C05452=1014.580,211.144,368.499,168.044,54.073,160.186
C05453=1014.586,211.393,368.475,168.049,54.063,160.185
C05454=1014.591,211.642,368.450,168.054,54.053,160.184
C05455=1014.596,211.890,368.426,168.058,54.042,160.182
C05456=1014.601,212.139,368.401,168.063,54.032,160.181
C05457=1014.606,212.388,368.377,168.067,54.022,160.180
C05458=1014.613,212.637,368.352,168.072,54.012,160.179
C05459=1014.618,212.885,368.328,168.076,54.002,160.178
C05460=1014.622,213.134,368.303,168.081,53.992,160.176
C05461=1014.628,213.383,368.278,168.084,53.982,160.175
C05462=1014.633,213.631,368.254,168.089,53.972,160.174
C05463=1014.639,213.881,368.230,168.094,53.962,160.173
C05464=1014.644,214.129,368.205,168.098,53.952,160.172
C05465=1014.649,214.378,368.180,168.103,53.942,160.171
C05466=1014.654,214.626,368.155,168.108,53.932,160.169
C05467=1014.660,214.875,368.131,168.113,53.922,160.168
C05468=1014.666,215.124,368.107,168.116,53.913,160.167
C05469=1014.670,215.373,368.082,168.121,53.902,160.166
C05470=1014.676,215.622,368.057,168.126,53.892,160.165
C05471=1014.682,215.870,368.032,168.130,53.883,160.164
C05472=1014.687,216.119,368.008,168.135,53.872,160.162
C05473=1014.691,216.367,367.983,168.140,53.863,160.161
C05474=1014.697,216.617,367.958,168.144,53.853,160.160
C05475=1014.703,216.865,367.933,168.148,53.843,160.159
C05476=1014.708,217.113,367.909,168.153,53.833,160.158
C05477=1014.714,217.363,367.885,168.158,53.823,160.157
C05478=1014.719,217.612,367.860,168.163,53.814,160.156
C05479=1014.724,217.859,367.835,168.166,53.803,160.154
C05480=1014.730,218.108,367.810,168.171,53.794,160.153
C05481=1014.735,218.355,367.785,168.176,53.784,160.152
C05482=1014.740,218.600,367.761,168.179,53.775,160.151
C05483=1014.745,218.846,367.736,168.184,53.765,160.150
C05484=1014.750,219.092,367.711,168.188,53.756,160.149
C05485=1014.756,219.338,367.686,168.193,53.746,160.147
C05486=1014.761,219.584,367.660,168.197,53.737,160.147
C05487=1014.766,219.829,367.636,168.202,53.728,160.145
C05488=1014.771,220.075,367.611,168.206,53.718,160.144
C05489=1014.777,220.324,367.587,168.211,53.709,160.143
C05490=1014.782,220.573,367.561,168.216,53.699,160.142
C05491=1014.787,220.821,367.537,168.220,53.690,160.141
C05492=1014.793,221.070,367.511,168.225,53.680,160.140
C05493=1014.798,221.318,367.486,168.230,53.670,160.139
C05494=1014.803,221.568,367.461,168.234,53.661,160.138
C05495=1014.809,221.816,367.436,168.238,53.651,160.137
C05496=1014.814,222.065,367.410,168.243,53.641,160.136
C05497=1014.820,222.313,367.385,168.247,53.632,160.134
C05498=1014.825,222.562,367.360,168.252,53.622,160.133
C05499=1014.831,222.811,367.335,168.257,53.614,160.132
C05500=1014.835,223.059,367.310,168.261,53.604,160.131
C05501=1014.842,223.308,367.284,168.266,53.594,160.130
C05502=1014.846,223.557,367.260,168.270,53.585,160.129
C05503=1014.852,223.806,367.234,168.275,53.575,160.128
C05504=1014.857,224.054,367.209,168.279,53.566,160.127
C05505=1014.862,224.303,367.183,168.285,53.557,160.126
C05506=1014.868,224.551,367.158,168.288,53.548,160.125
C05507=1014.873,224.800,367.132,168.293,53.538,160.124
C05508=1014.880,225.049,367.107,168.298,53.528,160.123
C05509=1014.884,225.298,367.082,168.303,53.520,160.122
C05510=1014.890,225.547,367.057,168.308,53.510,160.121
C05511=1014.895,225.795,367.031,168.312,53.501,160.120
C05512=1014.902,226.044,367.006,168.317,53.492,160.119
C05513=1014.906,226.292,366.980,168.321,53.483,160.118
C05514=1014.912,226.541,366.955,168.326,53.473,160.117
C05515=1014.916,226.790,366.930,168.330,53.464,160.116
C05516=1014.922,227.039,366.904,168.335,53.455,160.115
C05517=1014.928,227.287,366.878,168.340,53.446,160.114
C05518=1014.933,227.536,366.853,168.343,53.437,160.112
C05519=1014.938,227.785,366.827,168.349,53.428,160.112
C05520=1014.943,228.033,366.801,168.353,53.419,160.110
C05521=1014.949,228.282,366.776,168.358,53.410,160.110
C05522=1014.955,228.531,366.750,168.362,53.400,160.108
C05523=1014.960,228.779,366.725,168.368,53.392,160.108
C05524=1014.965,229.028,366.699,168.372,53.382,160.106
C05525=1014.970,229.276,366.673,168.376,53.374,160.105
C05526=1014.977,229.524,366.647,168.381,53.365,160.105
C05527=1014.982,229.773,366.621,168.385,53.355,160.103
C05528=1014.987,230.021,366.595,168.391,53.347,160.103
C05529=1014.992,230.270,366.570,168.395,53.338,160.102
C05530=1014.998,230.519,366.544,168.399,53.329,160.101
C05531=1015.003,230.768,366.518,168.405,53.320,160.100
C05532=1015.009,231.016,366.491,168.409,53.311,160.099
C05533=1015.014,231.265,366.465,168.413,53.303,160.098
C05534=1015.019,231.513,366.440,168.418,53.293,160.097
C05535=1015.024,231.762,366.414,168.423,53.284,160.096
C05536=1015.030,232.011,366.388,168.427,53.276,160.095
C05537=1015.035,232.259,366.362,168.432,53.267,160.094
C05538=1015.040,232.508,366.336,168.437,53.258,160.093
C05539=1015.046,232.757,366.310,168.441,53.249,160.092
C05540=1015.051,233.004,366.284,168.445,53.241,160.091
C05541=1015.057,233.246,366.258,168.450,53.232,160.090
C05542=1015.062,233.488,366.233,168.454,53.224,160.089
C05543=1015.068,233.730,366.208,168.460,53.215,160.088
C05544=1015.072,233.972,366.182,168.465,53.207,160.088
C05545=1015.078,234.213,366.157,168.469,53.198,160.087
C05546=1015.083,234.455,366.132,168.474,53.190,160.086
C05547=1015.089,234.697,366.107,168.478,53.181,160.085
C05548=1015.094,234.938,366.082,168.483,53.173,160.084
C05549=1015.100,235.187,366.055,168.487,53.164,160.083
C05550=1015.105,235.436,366.029,168.491,53.156,160.082
C05551=1015.111,235.684,366.003,168.497,53.147,160.081
C05552=1015.116,235.933,365.977,168.501,53.138,160.080
C05553=1015.121,236.181,365.951,168.506,53.130,160.079
C05554=1015.127,236.430,365.925,168.510,53.121,160.078
C05555=1015.132,236.679,365.899,168.515,53.113,160.077
C05556=1015.138,236.927,365.872,168.520,53.104,160.076
C05557=1015.144,237.176,365.846,168.525,53.095,160.076
C05558=1015.149,237.424,365.819,168.530,53.087,160.075
C05559=1015.154,237.673,365.794,168.534,53.079,160.074
C05560=1015.159,237.921,365.767,168.538,53.070,160.073
C05561=1015.165,238.170,365.740,168.544,53.061,160.072
C05562=1015.171,238.419,365.714,168.548,53.053,160.071
C05563=1015.176,238.667,365.687,168.553,53.044,160.070
C05564=1015.182,238.915,365.661,168.558,53.037,160.070
C05565=1015.187,239.164,365.635,168.562,53.028,160.069
C05566=1015.193,239.412,365.608,168.567,53.020,160.068
C05567=1015.198,239.661,365.581,168.572,53.012,160.067
C05568=1015.204,239.909,365.555,168.576,53.003,160.066
C05569=1015.209,240.158,365.529,168.582,52.994,160.065
C05570=1015.214,240.407,365.501,168.587,52.987,160.064
C05571=1015.220,240.655,365.475,168.591,52.978,160.064
C05572=1015.226,240.903,365.448,168.596,52.970,160.063
C05573=1015.230,241.153,365.422,168.600,52.962,160.062
C05574=1015.236,241.401,365.395,168.605,52.953,160.061
C05575=1015.242,241.649,365.368,168.610,52.946,160.060
C05576=1015.248,241.898,365.342,168.614,52.937,160.059
C05577=1015.253,242.146,365.314,168.619,52.929,160.059
C05578=1015.258,242.394,365.288,168.624,52.921,160.058
C05579=1015.264,242.642,365.261,168.629,52.913,160.057
C05580=1015.269,242.891,365.234,168.633,52.905,160.056
C05581=1015.275,243.139,365.208,168.638,52.897,160.055
C05582=1015.280,243.388,365.180,168.643,52.888,160.054
C05583=1015.285,243.636,365.154,168.648,52.880,160.054
C05584=1015.290,243.885,365.126,168.653,52.873,160.053
C05585=1015.295,244.134,365.099,168.657,52.864,160.052
C05586=1015.301,244.382,365.073,168.662,52.856,160.051
C05587=1015.306,244.631,365.045,168.667,52.849,160.051
C05588=1015.312,244.879,365.019,168.672,52.841,160.050
C05589=1015.317,245.127,364.991,168.676,52.832,160.049
C05590=1015.322,245.376,364.963,168.681,52.825,160.048
C05591=1015.328,245.624,364.937,168.686,52.817,160.047
C05592=1015.333,245.873,364.910,168.691,52.809,160.047
C05593=1015.339,246.121,364.883,168.696,52.801,160.046
C05594=1015.344,246.370,364.856,168.701,52.793,160.045
C05595=1015.350,246.619,364.827,168.705,52.785,160.044
C05596=1015.356,246.867,364.801,168.710,52.778,160.044
C05597=1015.361,247.116,364.773,168.715,52.770,160.043
C05598=1015.367,247.364,364.747,168.719,52.761,160.042
C05599=1015.372,247.612,364.719,168.724,52.754,160.041
C05600=1015.378,247.861,364.692,168.729,52.746,160.040
C05601=1015.383,248.098,364.666,168.734,52.738,160.040
C05602=1015.388,248.338,364.640,168.739,52.731,160.039
C05603=1015.393,248.576,364.614,168.743,52.724,160.038
C05604=1015.398,248.814,364.588,168.747,52.716,160.038
C05605=1015.404,249.052,364.561,168.752,52.708,160.037
C05606=1015.409,249.290,364.535,168.756,52.701,160.036
C05607=1015.414,249.529,364.508,168.762,52.694,160.036
C05608=1015.419,249.768,364.483,168.767,52.686,160.035
C05609=1015.425,250.015,364.455,168.771,52.679,160.034
C05610=1015.430,250.264,364.428,168.776,52.671,160.033
C05611=1015.437,250.512,364.400,168.781,52.663,160.033
C05612=1015.442,250.761,364.373,168.786,52.656,160.032
C05613=1015.447,251.010,364.346,168.791,52.648,160.031
C05614=1015.453,251.257,364.319,168.796,52.640,160.030
C05615=1015.458,251.506,364.291,168.801,52.632,160.030
C05616=1015.465,251.755,364.264,168.806,52.625,160.029
C05617=1015.470,252.003,364.236,168.810,52.617,160.028
C05618=1015.475,252.251,364.208,168.815,52.610,160.027
C05619=1015.481,252.500,364.182,168.820,52.602,160.027
C05620=1015.487,252.748,364.153,168.825,52.595,160.026
C05621=1015.493,252.997,364.127,168.830,52.587,160.026
C05622=1015.498,253.245,364.099,168.835,52.579,160.025
C05623=1015.504,253.494,364.071,168.840,52.572,160.024
C05624=1015.510,253.742,364.044,168.844,52.564,160.023
C05625=1015.515,253.991,364.017,168.849,52.556,160.023
C05626=1015.521,254.239,363.988,168.854,52.549,160.022
C05627=1015.527,254.488,363.962,168.859,52.542,160.021
C05628=1015.532,254.736,363.934,168.864,52.534,160.021
C05629=1015.539,254.984,363.906,168.869,52.526,160.020
C05630=1015.544,255.233,363.879,168.874,52.519,160.019
C05631=1015.549,255.481,363.851,168.879,52.512,160.019
C05632=1015.555,255.730,363.824,168.884,52.504,160.018
C05633=1015.561,255.978,363.796,168.889,52.496,160.017
C05634=1015.567,256.226,363.768,168.894,52.489,160.017
C05635=1015.572,256.475,363.741,168.899,52.482,160.016
C05636=1015.578,256.723,363.713,168.903,52.474,160.015
C05637=1015.584,256.972,363.685,168.909,52.467,160.015
C05638=1015.590,257.220,363.657,168.914,52.460,160.014
C05639=1015.595,257.469,363.630,168.919,52.452,160.013
C05640=1015.601,257.717,363.602,168.924,52.445,160.013
C05641=1015.607,257.965,363.574,168.929,52.437,160.012
C05642=1015.613,258.213,363.546,168.933,52.430,160.011
C05643=1015.618,258.462,363.519,168.939,52.423,160.011
C05644=1015.624,258.711,363.491,168.944,52.415,160.010
C05645=1015.631,258.958,363.464,168.949,52.408,160.009
C05646=1015.636,259.207,363.435,168.954,52.400,160.009
C05647=1015.643,259.455,363.408,168.959,52.394,160.008
C05648=1015.648,259.703,363.380,168.964,52.386,160.007
C05649=1015.654,259.952,363.352,168.969,52.379,160.007
C05650=1015.659,260.200,363.324,168.974,52.372,160.006
C05651=1015.665,260.449,363.295,168.979,52.365,160.006
C05652=1015.670,260.697,363.267,168.984,52.358,160.005
C05653=1015.676,260.945,363.239,168.988,52.351,160.004
C05654=1015.682,261.193,363.211,168.994,52.343,160.004
C05655=1015.688,261.442,363.182,168.999,52.336,160.003
C05656=1015.693,261.690,363.154,169.003,52.330,160.003
C05657=1015.699,261.938,363.126,169.009,52.323,160.002
C05658=1015.704,262.187,363.097,169.014,52.315,160.001
C05659=1015.710,262.435,363.069,169.018,52.308,160.001
C05660=1015.715,262.683,363.041,169.024,52.301,160.000
C05661=1015.721,262.921,363.014,169.028,52.295,160.000
C05662=1015.727,263.158,362.986,169.034,52.288,159.999
C05663=1015.732,263.396,362.959,169.038,52.281,159.999
C05664=1015.737,263.633,362.932,169.043,52.274,159.998
C05665=1015.743,263.870,362.905,169.049,52.268,159.998
C05666=1015.748,264.108,362.878,169.053,52.261,159.997
C05667=1015.754,264.345,362.851,169.058,52.255,159.997
C05668=1015.760,264.582,362.823,169.063,52.248,159.996
C05669=1015.765,264.830,362.795,169.067,52.241,159.995
C05670=1015.771,265.079,362.767,169.073,52.234,159.995
C05671=1015.777,265.326,362.738,169.077,52.228,159.994
C05672=1015.783,265.575,362.710,169.083,52.221,159.994
C05673=1015.788,265.824,362.680,169.088,52.214,159.993
C05674=1015.794,266.072,362.652,169.093,52.207,159.993
C05675=1015.799,266.320,362.624,169.098,52.200,159.992
C05676=1015.806,266.569,362.595,169.103,52.193,159.992
C05677=1015.811,266.817,362.567,169.108,52.186,159.991
C05678=1015.817,267.065,362.537,169.114,52.179,159.991
C05679=1015.823,267.314,362.509,169.119,52.173,159.990
C05680=1015.828,267.561,362.480,169.124,52.166,159.990
C05681=1015.834,267.810,362.452,169.129,52.160,159.989
C05682=1015.840,268.058,362.423,169.134,52.153,159.989
C05683=1015.846,268.307,362.393,169.140,52.146,159.988
C05684=1015.851,268.555,362.365,169.144,52.139,159.987
C05685=1015.857,268.803,362.336,169.150,52.132,159.987
C05686=1015.863,269.052,362.308,169.154,52.126,159.987
C05687=1015.868,269.299,362.279,169.160,52.119,159.986
C05688=1015.875,269.547,362.250,169.164,52.113,159.985
C05689=1015.880,269.796,362.220,169.170,52.106,159.985
C05690=1015.886,270.045,362.192,169.175,52.100,159.985
C05691=1015.892,270.292,362.163,169.180,52.093,159.984
C05692=1015.897,270.540,362.133,169.185,52.087,159.984
C05693=1015.903,270.789,362.104,169.191,52.080,159.983
C05694=1015.909,271.037,362.076,169.196,52.073,159.983
C05695=1015.915,271.286,362.046,169.201,52.067,159.982
C05696=1015.921,271.533,362.018,169.207,52.060,159.982
C05697=1015.926,271.782,361.988,169.211,52.054,159.981
C05698=1015.932,272.030,361.959,169.217,52.047,159.981
C05699=1015.939,272.278,361.930,169.222,52.041,159.980
C05700=1015.944,272.527,361.901,169.228,52.034,159.980
C05701=1015.949,272.774,361.872,169.232,52.028,159.979
C05702=1015.955,273.023,361.843,169.238,52.021,159.979
C05703=1015.961,273.271,361.814,169.242,52.015,159.978
C05704=1015.967,273.519,361.784,169.248,52.009,159.978
C05705=1015.973,273.768,361.755,169.253,52.002,159.978
C05706=1015.978,274.016,361.725,169.259,51.996,159.977
C05707=1015.985,274.264,361.696,169.264,51.990,159.977
C05708=1015.990,274.513,361.667,169.269,51.983,159.976
C05709=1015.996,274.761,361.638,169.274,51.977,159.976
C05710=1016.001,275.008,361.609,169.280,51.970,159.975
C05711=1016.008,275.257,361.579,169.285,51.964,159.975
C05712=1016.013,275.505,361.550,169.291,51.958,159.975
C05713=1016.020,275.753,361.520,169.295,51.951,159.974
C05714=1016.026,276.001,361.491,169.301,51.945,159.974
C05715=1016.031,276.249,361.461,169.306,51.939,159.974
C05716=1016.037,276.498,361.432,169.310,51.933,159.973
C05717=1016.043,276.746,361.403,169.316,51.926,159.973
C05718=1016.049,276.994,361.372,169.321,51.920,159.972
C05719=1016.054,277.242,361.343,169.327,51.914,159.972
C05720=1016.060,277.490,361.313,169.332,51.908,159.972
C05721=1016.066,277.729,361.285,169.337,51.902,159.971
C05722=1016.071,277.970,361.256,169.342,51.896,159.971
C05723=1016.077,278.209,361.227,169.348,51.890,159.970
C05724=1016.082,278.448,361.198,169.353,51.884,159.970
C05725=1016.089,278.688,361.170,169.358,51.878,159.970
C05726=1016.094,278.927,361.141,169.363,51.872,159.969
C05727=1016.100,279.167,361.112,169.368,51.867,159.969
C05728=1016.105,279.406,361.084,169.373,51.861,159.968
C05729=1016.111,279.655,361.054,169.379,51.854,159.968
C05730=1016.117,279.903,361.024,169.383,51.849,159.968
C05731=1016.123,280.151,360.994,169.389,51.842,159.967
C05732=1016.129,280.399,360.964,169.394,51.836,159.967
C05733=1016.134,280.647,360.934,169.400,51.830,159.967
C05734=1016.141,280.895,360.904,169.405,51.824,159.966
C05735=1016.147,281.144,360.875,169.410,51.818,159.966
C05736=1016.153,281.391,360.844,169.416,51.812,159.966
C05737=1016.158,281.640,360.815,169.421,51.806,159.965
C05738=1016.165,281.887,360.785,169.427,51.800,159.965
C05739=1016.170,282.136,360.755,169.432,51.794,159.965
C05740=1016.176,282.384,360.725,169.437,51.788,159.964
C05741=1016.182,282.633,360.695,169.443,51.783,159.964
C05742=1016.189,282.880,360.665,169.448,51.777,159.964
C05743=1016.195,283.128,360.635,169.454,51.771,159.963
C05744=1016.200,283.377,360.605,169.459,51.765,159.963
C05745=1016.206,283.624,360.575,169.465,51.758,159.963
C05746=1016.212,283.872,360.545,169.470,51.753,159.962
C05747=1016.219,284.121,360.515,169.475,51.747,159.962
C05748=1016.224,284.369,360.485,169.481,51.741,159.962
C05749=1016.230,284.617,360.454,169.486,51.735,159.961
C05750=1016.236,284.865,360.424,169.492,51.729,159.961
C05751=1016.242,285.114,360.394,169.498,51.724,159.961
C05752=1016.248,285.361,360.364,169.503,51.718,159.961
C05753=1016.254,285.609,360.333,169.508,51.712,159.960
C05754=1016.260,285.857,360.304,169.514,51.707,159.960
C05755=1016.267,286.105,360.273,169.519,51.701,159.960
C05756=1016.273,286.353,360.243,169.525,51.695,159.960
C05757=1016.278,286.601,360.212,169.530,51.689,159.959
C05758=1016.284,286.849,360.182,169.535,51.683,159.959
C05759=1016.291,287.097,360.151,169.541,51.678,159.959
C05760=1016.296,287.345,360.121,169.546,51.672,159.958
C05761=1016.302,287.593,360.090,169.552,51.667,159.958
C05762=1016.309,287.841,360.060,169.558,51.661,159.958
C05763=1016.315,288.089,360.029,169.563,51.655,159.958
C05764=1016.320,288.337,359.999,169.568,51.650,159.957
C05765=1016.326,288.586,359.968,169.574,51.644,159.957
C05766=1016.332,288.834,359.937,169.579,51.638,159.957
C05767=1016.338,289.082,359.907,169.586,51.633,159.957
C05768=1016.344,289.330,359.876,169.591,51.627,159.957
C05769=1016.350,289.578,359.846,169.596,51.622,159.956
C05770=1016.356,289.825,359.815,169.602,51.616,159.956
C05771=1016.362,290.074,359.784,169.607,51.610,159.956
C05772=1016.368,290.321,359.754,169.613,51.605,159.955
C05773=1016.375,290.570,359.723,169.619,51.599,159.955
C05774=1016.380,290.818,359.693,169.624,51.594,159.955
C05775=1016.387,291.065,359.662,169.630,51.588,159.955
C05776=1016.393,291.314,359.631,169.636,51.583,159.955
C05777=1016.398,291.562,359.600,169.641,51.578,159.955
C05778=1016.405,291.810,359.569,169.646,51.572,159.954
C05779=1016.411,292.057,359.538,169.653,51.566,159.954
C05780=1016.417,292.306,359.508,169.658,51.561,159.954
C05781=1016.423,292.551,359.477,169.663,51.556,159.954
C05782=1016.429,292.797,359.446,169.669,51.551,159.953
C05783=1016.435,293.043,359.416,169.675,51.545,159.953
C05784=1016.441,293.289,359.384,169.681,51.540,159.953
C05785=1016.446,293.534,359.353,169.686,51.535,159.953
C05786=1016.453,293.779,359.322,169.691,51.530,159.953
C05787=1016.458,294.026,359.292,169.697,51.524,159.953
C05788=1016.464,294.272,359.260,169.702,51.519,159.952
C05789=1016.470,294.519,359.229,169.708,51.514,159.952
C05790=1016.476,294.767,359.197,169.714,51.509,159.952
C05791=1016.482,295.015,359.167,169.719,51.503,159.952
C05792=1016.488,295.263,359.135,169.725,51.498,159.952
C05793=1016.493,295.511,359.103,169.731,51.493,159.952
C05794=1016.500,295.759,359.072,169.736,51.488,159.951
C05795=1016.505,296.007,359.041,169.742,51.482,159.951
C05796=1016.512,296.255,359.009,169.748,51.478,159.951
C05797=1016.518,296.503,358.977,169.754,51.472,159.951
C05798=1016.524,296.750,358.946,169.759,51.467,159.951
C05799=1016.530,296.999,358.915,169.765,51.462,159.951
C05800=1016.536,297.246,358.884,169.770,51.457,159.951
C05801=1016.542,297.494,358.852,169.777,51.452,159.951
C05802=1016.549,297.742,358.820,169.782,51.447,159.951
C05803=1016.554,297.990,358.789,169.788,51.442,159.950
C05804=1016.561,298.238,358.757,169.793,51.437,159.950
C05805=1016.567,298.486,358.725,169.799,51.431,159.950
C05806=1016.572,298.733,358.694,169.805,51.427,159.950
C05807=1016.579,298.981,358.662,169.811,51.421,159.950
C05808=1016.585,299.229,358.630,169.816,51.416,159.950
C05809=1016.591,299.477,358.599,169.823,51.411,159.950
C05810=1016.597,299.725,358.567,169.828,51.406,159.950
C05811=1016.604,299.973,358.536,169.834,51.401,159.949
C05812=1016.610,300.221,358.504,169.840,51.396,159.950
C05813=1016.616,300.468,358.472,169.846,51.391,159.949
C05814=1016.622,300.716,358.440,169.852,51.387,159.949
C05815=1016.628,300.964,358.409,169.857,51.381,159.949
C05816=1016.634,301.212,358.377,169.863,51.376,159.949
C05817=1016.640,301.460,358.345,169.869,51.371,159.949
C05818=1016.647,301.708,358.314,169.875,51.366,159.949
C05819=1016.653,301.956,358.282,169.880,51.362,159.949
C05820=1016.659,302.204,358.250,169.887,51.356,159.949
C05821=1016.665,302.452,358.218,169.893,51.352,159.949
C05822=1016.672,302.699,358.187,169.898,51.347,159.949
C05823=1016.678,302.947,358.155,169.905,51.342,159.949
C05824=1016.684,303.195,358.123,169.910,51.337,159.949
C05825=1016.690,303.443,358.091,169.916,51.332,159.949
C05826=1016.697,303.690,358.059,169.921,51.327,159.948
C05827=1016.703,303.939,358.027,169.928,51.322,159.949
C05828=1016.709,304.187,357.995,169.934,51.318,159.949
C05829=1016.716,304.435,357.963,169.939,51.313,159.948
C05830=1016.722,304.682,357.931,169.946,51.308,159.948
C05831=1016.729,304.929,357.900,169.952,51.303,159.948
C05832=1016.735,305.178,357.868,169.957,51.298,159.948
C05833=1016.742,305.425,357.835,169.963,51.294,159.948
C05834=1016.748,305.673,357.803,169.970,51.288,159.948
C05835=1016.755,305.920,357.771,169.975,51.284,159.948
C05836=1016.761,306.169,357.739,169.981,51.279,159.948
C05837=1016.767,306.417,357.707,169.988,51.274,159.948
C05838=1016.774,306.664,357.675,169.993,51.269,159.948
C05839=1016.780,306.912,357.643,169.999,51.265,159.948
C05840=1016.787,307.160,357.611,170.005,51.260,159.948
C05841=1016.793,307.422,357.577,170.011,51.255,159.948
C05842=1016.800,307.682,357.543,170.018,51.250,159.948
C05843=1016.807,307.944,357.509,170.025,51.245,159.948
C05844=1016.814,308.206,357.475,170.030,51.240,159.948
C05845=1016.821,308.453,357.443,170.037,51.235,159.948
C05846=1016.827,308.701,357.410,170.043,51.231,159.948
C05847=1016.834,308.949,357.379,170.049,51.226,159.948
C05848=1016.840,309.196,357.346,170.056,51.221,159.948
C05849=1016.847,309.444,357.315,170.061,51.217,159.948
C05850=1016.853,309.692,357.282,170.067,51.212,159.948
C05851=1016.859,309.940,357.248,170.073,51.208,159.948
C05852=1016.865,310.187,357.216,170.080,51.203,159.948
C05853=1016.871,310.435,357.183,170.086,51.199,159.948
C05854=1016.878,310.683,357.150,170.092,51.194,159.948
C05855=1016.884,310.930,357.118,170.098,51.190,159.949
C05856=1016.890,311.179,357.084,170.104,51.186,159.949
C05857=1016.896,311.426,357.051,170.109,51.182,159.949
C05858=1016.903,311.674,357.018,170.116,51.177,159.949
C05859=1016.909,311.921,356.985,170.122,51.173,159.949
C05860=1016.916,312.169,356.952,170.128,51.168,159.949
C05861=1016.921,312.416,356.919,170.134,51.164,159.949
C05862=1016.928,312.664,356.886,170.140,51.159,159.949
C05863=1016.934,312.912,356.853,170.147,51.155,159.949
C05864=1016.941,313.160,356.820,170.153,51.151,159.949
C05865=1016.947,313.408,356.787,170.159,51.147,159.950
C05866=1016.953,313.655,356.753,170.165,51.143,159.950
C05867=1016.959,313.902,356.721,170.172,51.138,159.950
C05868=1016.966,314.151,356.688,170.178,51.134,159.950
C05869=1016.972,314.398,356.655,170.184,51.130,159.950
C05870=1016.979,314.645,356.621,170.190,51.126,159.950
C05871=1016.984,314.893,356.588,170.196,51.121,159.950
C05872=1016.991,315.141,356.555,170.203,51.116,159.950
C05873=1016.998,315.388,356.521,170.209,51.113,159.950
C05874=1017.004,315.636,356.489,170.215,51.108,159.950
C05875=1017.011,315.884,356.456,170.221,51.104,159.951
C05876=1017.017,316.132,356.422,170.228,51.100,159.951
C05877=1017.023,316.379,356.389,170.234,51.096,159.951
C05878=1017.031,316.627,356.355,170.240,51.092,159.951
C05879=1017.037,316.874,356.322,170.246,51.088,159.951
C05880=1017.043,317.123,356.289,170.253,51.083,159.952
C05881=1017.050,317.370,356.255,170.259,51.079,159.952
C05882=1017.056,317.618,356.222,170.265,51.075,159.952
C05883=1017.063,317.865,356.188,170.271,51.071,159.952
C05884=1017.069,318.113,356.156,170.278,51.067,159.952
C05885=1017.076,318.361,356.121,170.284,51.063,159.952
C05886=1017.082,318.609,356.089,170.290,51.058,159.952
C05887=1017.089,318.856,356.055,170.297,51.054,159.953
C05888=1017.096,319.103,356.021,170.304,51.050,159.953
C05889=1017.102,319.352,355.988,170.310,51.047,159.953
C05890=1017.109,319.599,355.954,170.316,51.042,159.953
C05891=1017.116,319.846,355.920,170.323,51.038,159.953
C05892=1017.122,320.094,355.888,170.329,51.034,159.954
C05893=1017.129,320.342,355.854,170.335,51.030,159.954
C05894=1017.135,320.589,355.820,170.341,51.026,159.954
C05895=1017.142,320.837,355.787,170.348,51.022,159.954
C05896=1017.149,321.085,355.753,170.355,51.018,159.954
C05897=1017.156,321.332,355.719,170.361,51.014,159.954
C05898=1017.162,321.580,355.685,170.368,51.010,159.955
C05899=1017.169,321.827,355.652,170.374,51.006,159.955
C05900=1017.176,322.075,355.618,170.380,51.002,159.955
C05901=1017.183,322.342,355.581,170.387,50.998,159.955
C05902=1017.190,322.608,355.545,170.394,50.994,159.956
C05903=1017.198,322.875,355.509,170.402,50.989,159.956
C05904=1017.205,323.142,355.473,170.409,50.985,159.956
C05905=1017.212,323.389,355.439,170.415,50.981,159.956
C05906=1017.219,323.638,355.406,170.421,50.978,159.957
C05907=1017.225,323.885,355.372,170.429,50.974,159.957
C05908=1017.232,324.133,355.338,170.435,50.970,159.957
C05909=1017.239,324.380,355.304,170.441,50.966,159.957
C05910=1017.246,324.628,355.270,170.448,50.962,159.958
C05911=1017.253,324.876,355.236,170.454,50.958,159.958
C05912=1017.260,325.123,355.202,170.461,50.954,159.958
C05913=1017.267,325.371,355.168,170.468,50.950,159.958
C05914=1017.274,325.618,355.135,170.474,50.946,159.959
C05915=1017.281,325.866,355.099,170.480,50.943,159.959
C05916=1017.288,326.113,355.066,170.488,50.939,159.959
C05917=1017.295,326.360,355.032,170.494,50.935,159.960
C05918=1017.301,326.608,354.998,170.500,50.931,159.960
C05919=1017.308,326.856,354.963,170.508,50.927,159.960
C05920=1017.315,327.103,354.929,170.514,50.924,159.960
C05921=1017.321,327.351,354.894,170.520,50.920,159.961
C05922=1017.328,327.599,354.859,170.528,50.917,159.961
C05923=1017.335,327.846,354.826,170.534,50.913,159.961
C05924=1017.342,328.093,354.791,170.540,50.909,159.962
C05925=1017.348,328.341,354.756,170.547,50.906,159.962
C05926=1017.356,328.588,354.722,170.554,50.902,159.962
C05927=1017.362,328.836,354.687,170.561,50.899,159.963
C05928=1017.369,329.083,354.652,170.567,50.895,159.963
C05929=1017.375,329.331,354.618,170.575,50.892,159.963
C05930=1017.383,329.578,354.583,170.581,50.888,159.964
C05931=1017.389,329.826,354.549,170.588,50.885,159.964
C05932=1017.396,330.074,354.514,170.595,50.881,159.964
C05933=1017.403,330.321,354.479,170.601,50.878,159.965
C05934=1017.410,330.569,354.445,170.608,50.874,159.965
C05935=1017.417,330.816,354.409,170.615,50.870,159.965
C05936=1017.424,331.063,354.375,170.622,50.867,159.966
C05937=1017.431,331.311,354.341,170.629,50.864,159.966
C05938=1017.437,331.559,354.305,170.636,50.860,159.967
C05939=1017.444,331.806,354.270,170.642,50.857,159.967
C05940=1017.451,332.054,354.236,170.649,50.854,159.967
C05941=1017.458,332.301,354.201,170.656,50.850,159.968
C05942=1017.465,332.548,354.166,170.663,50.846,159.968
C05943=1017.472,332.796,354.131,170.669,50.843,159.969
C05944=1017.478,333.043,354.096,170.677,50.840,159.969
C05945=1017.487,333.291,354.061,170.684,50.837,159.969
C05946=1017.493,333.538,354.026,170.690,50.833,159.970
C05947=1017.500,333.786,353.991,170.698,50.829,159.970
C05948=1017.507,334.033,353.956,170.704,50.826,159.971
C05949=1017.514,334.280,353.920,170.711,50.823,159.971
C05950=1017.520,334.528,353.885,170.718,50.820,159.971
C05951=1017.527,334.775,353.850,170.725,50.817,159.972
C05952=1017.535,335.023,353.815,170.732,50.813,159.972
C05953=1017.541,335.270,353.780,170.739,50.810,159.973
C05954=1017.548,335.517,353.744,170.746,50.807,159.973
C05955=1017.555,335.765,353.709,170.752,50.804,159.974
C05956=1017.563,336.013,353.673,170.760,50.800,159.974
C05957=1017.569,336.260,353.638,170.767,50.797,159.975
C05958=1017.576,336.507,353.603,170.773,50.794,159.975
C05959=1017.583,336.754,353.567,170.781,50.790,159.975
C05960=1017.590,337.002,353.531,170.788,50.787,159.976
C05961=1017.598,337.265,353.494,170.796,50.785,159.977
C05962=1017.606,337.527,353.457,170.803,50.781,159.977
C05963=1017.613,337.790,353.419,170.811,50.778,159.978
C05964=1017.620,338.052,353.381,170.818,50.774,159.978
C05965=1017.627,338.300,353.346,170.825,50.771,159.978
C05966=1017.635,338.547,353.310,170.832,50.768,159.979
C05967=1017.642,338.795,353.274,170.840,50.765,159.980
C05968=1017.649,339.042,353.238,170.846,50.762,159.980
C05969=1017.656,339.289,353.203,170.854,50.758,159.981
C05970=1017.663,339.536,353.167,170.861,50.756,159.981
C05971=1017.671,339.783,353.131,170.868,50.753,159.982
C05972=1017.678,340.031,353.096,170.875,50.749,159.982
C05973=1017.684,340.278,353.059,170.882,50.747,159.983
C05974=1017.691,340.526,353.024,170.890,50.743,159.983
C05975=1017.699,340.773,352.988,170.897,50.741,159.984
C05976=1017.706,341.020,352.952,170.903,50.738,159.984
C05977=1017.713,341.267,352.916,170.911,50.735,159.985
C05978=1017.719,341.515,352.880,170.918,50.732,159.985
C05979=1017.727,341.762,352.844,170.926,50.729,159.986
C05980=1017.734,342.009,352.808,170.933,50.726,159.986
C05981=1017.742,342.256,352.772,170.941,50.723,159.987
C05982=1017.748,342.504,352.735,170.947,50.720,159.988
C05983=1017.756,342.751,352.699,170.954,50.717,159.988
C05984=1017.764,342.998,352.663,170.962,50.715,159.989
C05985=1017.771,343.245,352.627,170.969,50.711,159.989
C05986=1017.778,343.493,352.590,170.977,50.709,159.990
C05987=1017.785,343.740,352.554,170.984,50.706,159.991
C05988=1017.792,343.987,352.518,170.992,50.703,159.991
C05989=1017.799,344.235,352.481,170.999,50.700,159.992
C05990=1017.806,344.482,352.445,171.007,50.697,159.992
C05991=1017.814,344.729,352.409,171.014,50.695,159.993
C05992=1017.821,344.977,352.372,171.021,50.692,159.994
C05993=1017.828,345.224,352.337,171.028,50.689,159.994
C05994=1017.836,345.471,352.300,171.035,50.686,159.995
C05995=1017.843,345.719,352.264,171.043,50.684,159.995
C05996=1017.850,345.966,352.227,171.050,50.681,159.996
C05997=1017.858,346.212,352.191,171.058,50.678,159.997
C05998=1017.865,346.460,352.155,171.065,50.676,159.997
C05999=1017.872,346.708,352.118,171.073,50.673,159.998
C06000=1017.880,346.954,352.081,171.080,50.671,159.999
C06001=1017.887,347.201,352.044,171.088,50.668,159.999
C06002=1017.894,347.449,352.008,171.095,50.665,160.000
C06003=1017.902,347.696,351.971,171.103,50.662,160.001
C06004=1017.909,347.943,351.934,171.110,50.660,160.001
C06005=1017.916,348.191,351.897,171.118,50.657,160.002
C06006=1017.924,348.438,351.861,171.125,50.655,160.003
C06007=1017.931,348.684,351.824,171.133,50.652,160.003
C06008=1017.938,348.932,351.787,171.140,50.649,160.004
C06009=1017.946,349.179,351.750,171.149,50.647,160.005
C06010=1017.953,349.426,351.712,171.156,50.645,160.005
C06011=1017.961,349.674,351.676,171.164,50.642,160.006
C06012=1017.968,349.921,351.639,171.172,50.639,160.007
C06013=1017.976,350.168,351.602,171.179,50.637,160.008
C06014=1017.983,350.415,351.565,171.187,50.634,160.008
C06015=1017.991,350.662,351.528,171.194,50.632,160.009
C06016=1017.998,350.909,351.490,171.202,50.629,160.010
C06017=1018.005,351.156,351.453,171.210,50.627,160.011
C06018=1018.013,351.404,351.417,171.218,50.624,160.011
C06019=1018.020,351.651,351.379,171.225,50.622,160.012
C06020=1018.028,351.898,351.342,171.233,50.620,160.013
C06021=1018.036,352.158,351.303,171.241,50.617,160.013
C06022=1018.044,352.417,351.264,171.249,50.615,160.014
C06023=1018.052,352.677,351.225,171.257,50.612,160.015
C06024=1018.060,352.937,351.185,171.266,50.610,160.016
C06025=1018.068,353.184,351.148,171.274,50.607,160.017
C06026=1018.075,353.431,351.111,171.281,50.605,160.017
C06027=1018.082,353.678,351.073,171.290,50.603,160.018
C06028=1018.090,353.925,351.036,171.297,50.600,160.019
C06029=1018.097,354.172,350.999,171.305,50.598,160.020
C06030=1018.105,354.420,350.961,171.313,50.595,160.021
C06031=1018.113,354.666,350.923,171.321,50.593,160.021
C06032=1018.121,354.913,350.886,171.329,50.591,160.022
C06033=1018.128,355.160,350.848,171.337,50.589,160.023
C06034=1018.135,355.407,350.811,171.344,50.586,160.024
C06035=1018.143,355.655,350.772,171.353,50.584,160.025
C06036=1018.151,355.902,350.735,171.361,50.582,160.026
C06037=1018.159,356.149,350.698,171.369,50.580,160.026
C06038=1018.166,356.395,350.659,171.377,50.578,160.027
C06039=1018.174,356.643,350.621,171.385,50.575,160.028
C06040=1018.181,356.890,350.584,171.392,50.573,160.029
C06041=1018.190,357.136,350.546,171.401,50.571,160.030
C06042=1018.197,357.384,350.508,171.409,50.569,160.031
C06043=1018.205,357.631,350.470,171.417,50.567,160.031
C06044=1018.212,357.878,350.433,171.425,50.565,160.032
C06045=1018.220,358.125,350.394,171.433,50.563,160.033
C06046=1018.228,358.371,350.356,171.441,50.561,160.034
C06047=1018.236,358.618,350.319,171.449,50.558,160.035
C06048=1018.244,358.865,350.280,171.457,50.556,160.036
C06049=1018.252,359.112,350.242,171.466,50.554,160.037
C06050=1018.260,359.360,350.204,171.473,50.552,160.038
C06051=1018.267,359.606,350.166,171.482,50.550,160.039
C06052=1018.275,359.854,350.127,171.490,50.548,160.040
C06053=1018.283,360.100,350.089,171.498,50.547,160.040
C06054=1018.290,360.347,350.051,171.506,50.544,160.041
C06055=1018.298,360.594,350.012,171.515,50.542,160.042
C06056=1018.305,360.841,349.973,171.523,50.541,160.043
C06057=1018.313,361.088,349.935,171.531,50.539,160.044
C06058=1018.321,361.334,349.896,171.539,50.537,160.045
C06059=1018.329,361.582,349.858,171.548,50.535,160.046
C06060=1018.337,361.829,349.819,171.556,50.533,160.047
C06061=1018.345,362.075,349.781,171.564,50.532,160.048
C06062=1018.353,362.323,349.742,171.573,50.529,160.049
C06063=1018.361,362.569,349.704,171.581,50.527,160.050
C06064=1018.369,362.816,349.666,171.590,50.526,160.051
C06065=1018.376,363.063,349.627,171.598,50.523,160.052
C06066=1018.384,363.310,349.587,171.606,50.522,160.053
C06067=1018.392,363.557,349.549,171.614,50.520,160.054
C06068=1018.400,363.803,349.511,171.623,50.518,160.055
C06069=1018.408,364.051,349.472,171.632,50.517,160.056
C06070=1018.416,364.297,349.433,171.640,50.514,160.057
C06071=1018.424,364.544,349.394,171.649,50.513,160.058
C06072=1018.432,364.791,349.356,171.656,50.511,160.059
C06073=1018.440,365.038,349.316,171.665,50.509,160.060
C06074=1018.449,365.285,349.278,171.674,50.508,160.061
C06075=1018.457,365.531,349.238,171.682,50.506,160.062
C06076=1018.464,365.778,349.200,171.691,50.504,160.063
C06077=1018.472,366.025,349.160,171.700,50.502,160.064
C06078=1018.480,366.272,349.122,171.709,50.501,160.065
C06079=1018.489,366.519,349.082,171.718,50.499,160.066
C06080=1018.497,366.766,349.044,171.726,50.497,160.067
C06081=1018.506,367.033,349.001,171.735,50.495,160.068
C06082=1018.515,367.300,348.959,171.745,50.494,160.070
C06083=1018.524,367.567,348.917,171.753,50.492,160.071
C06084=1018.533,367.834,348.874,171.764,50.491,160.072
C06085=1018.540,368.081,348.834,171.772,50.489,160.073
C06086=1018.549,368.328,348.795,171.781,50.487,160.074
C06087=1018.556,368.575,348.756,171.790,50.486,160.076
C06088=1018.565,368.822,348.716,171.799,50.484,160.077
C06089=1018.573,369.068,348.677,171.807,50.483,160.078
C06090=1018.581,369.315,348.637,171.816,50.481,160.079
C06091=1018.589,369.562,348.598,171.825,50.479,160.080
C06092=1018.597,369.809,348.558,171.834,50.478,160.081
C06093=1018.606,370.055,348.518,171.843,50.477,160.082
C06094=1018.614,370.302,348.478,171.852,50.475,160.083
C06095=1018.622,370.548,348.438,171.861,50.474,160.085
C06096=1018.630,370.795,348.399,171.870,50.473,160.086
C06097=1018.638,371.042,348.359,171.878,50.471,160.087
C06098=1018.647,371.288,348.320,171.887,50.470,160.088
C06099=1018.655,371.535,348.279,171.896,50.469,160.089
C06100=1018.663,371.781,348.240,171.905,50.467,160.091
C06101=1018.671,372.029,348.200,171.914,50.465,160.092
C06102=1018.680,372.275,348.160,171.923,50.464,160.093
C06103=1018.688,372.522,348.120,171.932,50.463,160.094
C06104=1018.696,372.768,348.080,171.941,50.462,160.095
C06105=1018.705,373.014,348.040,171.950,50.460,160.097
C06106=1018.713,373.262,348.000,171.959,50.459,160.098
C06107=1018.722,373.508,347.960,171.968,50.458,160.099
C06108=1018.730,373.755,347.920,171.977,50.457,160.100
C06109=1018.739,374.001,347.880,171.987,50.455,160.102
C06110=1018.747,374.248,347.840,171.996,50.454,160.103
C06111=1018.756,374.494,347.800,172.005,50.453,160.104
C06112=1018.764,374.741,347.760,172.014,50.452,160.105
C06113=1018.773,374.988,347.719,172.023,50.450,160.106
C06114=1018.782,375.234,347.679,172.032,50.449,160.108
C06115=1018.790,375.482,347.639,172.042,50.448,160.109
C06116=1018.799,375.727,347.599,172.052,50.447,160.111
C06117=1018.807,375.974,347.558,172.060,50.445,160.112
C06118=1018.815,376.221,347.517,172.070,50.444,160.113
C06119=1018.824,376.467,347.477,172.079,50.443,160.114
C06120=1018.833,376.714,347.436,172.088,50.442,160.116
C06121=1018.841,376.960,347.396,172.098,50.441,160.117
C06122=1018.849,377.207,347.355,172.107,50.440,160.118
C06123=1018.857,377.453,347.314,172.116,50.439,160.120
C06124=1018.867,377.700,347.274,172.126,50.438,160.121
C06125=1018.875,377.946,347.233,172.136,50.436,160.122
C06126=1018.883,378.193,347.192,172.145,50.436,160.124
C06127=1018.892,378.439,347.151,172.154,50.435,160.125
C06128=1018.901,378.686,347.110,172.164,50.434,160.127
C06129=1018.909,378.932,347.070,172.174,50.433,160.128
C06130=1018.918,379.179,347.029,172.183,50.432,160.129
C06131=1018.926,379.424,346.987,172.192,50.431,160.131
C06132=1018.935,379.671,346.946,172.202,50.430,160.132
C06133=1018.944,379.918,346.906,172.212,50.429,160.133
C06134=1018.952,380.164,346.865,172.221,50.428,160.135
C06135=1018.961,380.411,346.824,172.231,50.428,160.136
C06136=1018.970,380.657,346.782,172.241,50.426,160.138
C06137=1018.979,380.904,346.741,172.250,50.426,160.139
C06138=1018.988,381.149,346.700,172.260,50.424,160.141
C06139=1018.996,381.396,346.659,172.270,50.424,160.142
C06140=1019.005,381.643,346.617,172.279,50.423,160.143
C06141=1019.016,381.932,346.569,172.291,50.422,160.145
C06142=1019.026,382.222,346.521,172.302,50.421,160.147
C06143=1019.036,382.511,346.472,172.314,50.420,160.149
C06144=1019.047,382.801,346.424,172.326,50.419,160.150
C06145=1019.056,383.047,346.382,172.335,50.418,160.152
C06146=1019.065,383.293,346.340,172.345,50.417,160.153
C06147=1019.074,383.540,346.300,172.355,50.417,160.155
C06148=1019.083,383.786,346.258,172.365,50.416,160.156
C06149=1019.092,384.033,346.216,172.375,50.415,160.158
C06150=1019.101,384.279,346.175,172.385,50.414,160.159
C06151=1019.110,384.525,346.133,172.395,50.414,160.161
C06152=1019.120,384.771,346.092,172.405,50.413,160.163
C06153=1019.129,385.018,346.050,172.416,50.412,160.164
C06154=1019.137,385.264,346.008,172.425,50.411,160.166
C06155=1019.146,385.511,345.967,172.436,50.411,160.167
C06156=1019.155,385.757,345.925,172.445,50.410,160.169
C06157=1019.165,386.003,345.882,172.456,50.410,160.170
C06158=1019.174,386.249,345.841,172.465,50.409,160.172
C06159=1019.182,386.495,345.799,172.476,50.409,160.174
C06160=1019.192,386.742,345.756,172.486,50.409,160.175
C06161=1019.201,386.988,345.715,172.496,50.408,160.177
C06162=1019.210,387.235,345.673,172.507,50.407,160.178
C06163=1019.219,387.480,345.630,172.516,50.407,160.180
C06164=1019.228,387.727,345.589,172.527,50.406,160.181
C06165=1019.238,387.972,345.546,172.538,50.406,160.183
C06166=1019.247,388.219,345.504,172.547,50.405,160.185
C06167=1019.256,388.466,345.461,172.558,50.404,160.186
C06168=1019.265,388.711,345.419,172.569,50.404,160.188
C06169=1019.274,388.958,345.377,172.579,50.404,160.190
C06170=1019.284,389.204,345.334,172.589,50.404,160.192
C06171=1019.293,389.450,345.292,172.600,50.403,160.193
C06172=1019.301,389.696,345.249,172.610,50.403,160.195
C06173=1019.311,389.942,345.206,172.620,50.402,160.197
C06174=1019.320,390.188,345.163,172.631,50.402,160.198
C06175=1019.329,390.434,345.122,172.642,50.401,160.200
C06176=1019.339,390.681,345.079,172.653,50.401,160.202
C06177=1019.348,390.927,345.036,172.663,50.401,160.204
C06178=1019.358,391.173,344.993,172.673,50.400,160.205
C06179=1019.367,391.419,344.951,172.684,50.400,160.207
C06180=1019.377,391.666,344.908,172.695,50.400,160.209
C06181=1019.386,391.911,344.865,172.706,50.400,160.211
C06182=1019.395,392.157,344.821,172.716,50.399,160.212
C06183=1019.405,392.403,344.779,172.727,50.399,160.214
C06184=1019.414,392.650,344.736,172.738,50.399,160.216
C06185=1019.423,392.895,344.692,172.749,50.399,160.218
C06186=1019.433,393.142,344.650,172.760,50.399,160.219
C06187=1019.443,393.388,344.607,172.770,50.398,160.221
C06188=1019.452,393.633,344.563,172.781,50.398,160.223
C06189=1019.461,393.880,344.520,172.792,50.398,160.225
C06190=1019.471,394.125,344.477,172.803,50.398,160.227
C06191=1019.480,394.372,344.434,172.814,50.398,160.229
C06192=1019.490,394.618,344.390,172.825,50.397,160.230
C06193=1019.499,394.864,344.347,172.835,50.398,160.232
C06194=1019.509,395.109,344.304,172.846,50.398,160.234
C06195=1019.519,395.355,344.260,172.858,50.397,160.236
C06196=1019.528,395.602,344.217,172.869,50.397,160.238
C06197=1019.538,395.848,344.173,172.881,50.397,160.240
C06198=1019.548,396.093,344.130,172.892,50.397,160.242
C06199=1019.557,396.339,344.086,172.902,50.397,160.244
C06200=1019.567,396.585,344.042,172.914,50.397,160.246
C06201=1019.581,396.912,343.985,172.929,50.397,160.248
C06202=1019.593,397.240,343.926,172.943,50.397,160.251
C06203=1019.606,397.566,343.868,172.958,50.398,160.253
C06204=1019.620,397.894,343.810,172.973,50.398,160.256
C06205=1019.629,398.140,343.766,172.984,50.398,160.258
C06206=1019.639,398.386,343.722,172.997,50.398,160.260
C06207=1019.649,398.631,343.678,173.008,50.398,160.262
C06208=1019.659,398.877,343.634,173.019,50.398,160.264
C06209=1019.668,399.123,343.590,173.030,50.398,160.266
C06210=1019.678,399.369,343.545,173.042,50.399,160.268
C06211=1019.688,399.615,343.502,173.054,50.399,160.270
C06212=1019.698,399.861,343.458,173.065,50.399,160.272
C06213=1019.708,400.106,343.413,173.076,50.399,160.274
C06214=1019.718,400.352,343.369,173.088,50.399,160.276
C06215=1019.727,400.597,343.324,173.100,50.399,160.278
C06216=1019.738,400.843,343.280,173.111,50.400,160.280
C06217=1019.748,401.090,343.236,173.123,50.401,160.282
C06218=1019.757,401.335,343.191,173.135,50.401,160.285
C06219=1019.767,401.581,343.146,173.147,50.401,160.287
C06220=1019.777,401.826,343.101,173.158,50.401,160.289
C06221=1019.788,402.073,343.057,173.170,50.401,160.291
C06222=1019.797,402.318,343.013,173.182,50.402,160.293
C06223=1019.807,402.564,342.968,173.193,50.402,160.295
C06224=1019.817,402.810,342.922,173.206,50.402,160.297
C06225=1019.828,403.055,342.878,173.217,50.403,160.299
C06226=1019.837,403.301,342.833,173.230,50.403,160.302
C06227=1019.848,403.547,342.788,173.241,50.404,160.304
C06228=1019.858,403.792,342.743,173.254,50.404,160.306
C06229=1019.868,404.039,342.698,173.265,50.405,160.308
C06230=1019.879,404.283,342.653,173.278,50.405,160.310
C06231=1019.889,404.529,342.608,173.289,50.406,160.313
C06232=1019.899,404.775,342.563,173.302,50.406,160.315
C06233=1019.909,405.021,342.518,173.313,50.407,160.317
C06234=1019.920,405.266,342.473,173.326,50.407,160.319
C06235=1019.930,405.512,342.428,173.338,50.407,160.321
C06236=1019.940,405.757,342.382,173.350,50.408,160.324
C06237=1019.950,406.003,342.337,173.363,50.409,160.326
C06238=1019.961,406.249,342.293,173.376,50.409,160.328
C06239=1019.971,406.494,342.247,173.387,50.410,160.330
C06240=1019.982,406.739,342.201,173.400,50.410,160.333
C06241=1019.992,406.986,342.156,173.412,50.411,160.335
C06242=1020.003,407.231,342.110,173.424,50.412,160.337
C06243=1020.013,407.476,342.066,173.437,50.412,160.340
C06244=1020.024,407.722,342.020,173.449,50.413,160.342
C06245=1020.035,407.968,341.974,173.462,50.413,160.344
C06246=1020.045,408.213,341.928,173.475,50.414,160.347
C06247=1020.056,408.459,341.884,173.487,50.415,160.349
C06248=1020.067,408.705,341.838,173.500,50.416,160.351
C06249=1020.078,408.950,341.792,173.512,50.416,160.354
C06250=1020.088,409.196,341.746,173.525,50.417,160.356
C06251=1020.099,409.441,341.700,173.538,50.418,160.359
C06252=1020.110,409.686,341.653,173.551,50.418,160.361
C06253=1020.120,409.932,341.607,173.564,50.419,160.364
C06254=1020.130,410.178,341.561,173.576,50.420,160.366
C06255=1020.141,410.423,341.515,173.589,50.421,160.368
C06256=1020.152,410.668,341.468,173.602,50.422,160.371
C06257=1020.162,410.914,341.422,173.615,50.423,160.373
C06258=1020.173,411.160,341.377,173.628,50.424,160.376
C06259=1020.184,411.405,341.330,173.641,50.425,160.378
C06260=1020.195,411.650,341.284,173.654,50.426,160.381
C06261=1020.208,411.941,341.229,173.669,50.427,160.384
C06262=1020.220,412.231,341.174,173.685,50.427,160.387
C06263=1020.233,412.522,341.119,173.701,50.429,160.390
C06264=1020.246,412.813,341.064,173.716,50.430,160.393
C06265=1020.257,413.058,341.017,173.729,50.431,160.395
C06266=1020.269,413.303,340.970,173.743,50.432,160.398
C06267=1020.280,413.548,340.924,173.756,50.433,160.400
C06268=1020.290,413.793,340.877,173.769,50.434,160.403
C06269=1020.302,414.039,340.830,173.783,50.435,160.405
C06270=1020.312,414.285,340.783,173.797,50.435,160.408
C06271=1020.323,414.530,340.736,173.810,50.437,160.411
C06272=1020.334,414.775,340.690,173.823,50.438,160.413
C06273=1020.346,415.021,340.643,173.836,50.439,160.416
C06274=1020.357,415.265,340.595,173.850,50.440,160.419
C06275=1020.368,415.511,340.548,173.864,50.441,160.421
C06276=1020.379,415.756,340.501,173.877,50.443,160.424
C06277=1020.391,416.001,340.454,173.892,50.444,160.427
C06278=1020.401,416.247,340.406,173.905,50.445,160.429
C06279=1020.412,416.492,340.359,173.919,50.446,160.432
C06280=1020.424,416.737,340.312,173.932,50.447,160.435
C06281=1020.434,416.983,340.264,173.947,50.448,160.438
C06282=1020.446,417.228,340.217,173.960,50.450,160.440
C06283=1020.458,417.473,340.169,173.975,50.451,160.443
C06284=1020.469,417.719,340.121,173.988,50.452,160.446
C06285=1020.480,417.963,340.074,174.002,50.453,160.449
C06286=1020.491,418.209,340.026,174.016,50.455,160.451
C06287=1020.503,418.454,339.979,174.030,50.456,160.454
C06288=1020.515,418.699,339.931,174.045,50.457,160.457
C06289=1020.526,418.945,339.883,174.058,50.459,160.460
C06290=1020.538,419.190,339.835,174.073,50.460,160.463
C06291=1020.549,419.435,339.787,174.087,50.461,160.466
C06292=1020.560,419.680,339.739,174.101,50.463,160.468
C06293=1020.572,419.925,339.691,174.115,50.464,160.471
C06294=1020.584,420.170,339.644,174.130,50.466,160.474
C06295=1020.595,420.416,339.595,174.145,50.467,160.477
C06296=1020.607,420.660,339.547,174.158,50.469,160.480
C06297=1020.619,420.905,339.499,174.173,50.470,160.483
C06298=1020.630,421.150,339.451,174.188,50.471,160.486
C06299=1020.643,421.396,339.403,174.202,50.473,160.489
C06300=1020.654,421.641,339.354,174.217,50.474,160.492
C06301=1020.666,421.886,339.306,174.231,50.476,160.495
C06302=1020.677,422.131,339.257,174.246,50.477,160.498
C06303=1020.689,422.375,339.208,174.261,50.479,160.501
C06304=1020.701,422.621,339.160,174.276,50.480,160.504
C06305=1020.713,422.866,339.111,174.291,50.482,160.507
C06306=1020.725,423.110,339.063,174.305,50.484,160.510
C06307=1020.737,423.356,339.013,174.320,50.485,160.513
C06308=1020.749,423.601,338.966,174.335,50.487,160.516
C06309=1020.760,423.846,338.917,174.350,50.489,160.519
C06310=1020.772,424.091,338.867,174.365,50.490,160.522
C06311=1020.784,424.336,338.819,174.381,50.492,160.525
C06312=1020.796,424.581,338.769,174.396,50.493,160.528
C06313=1020.808,424.825,338.721,174.411,50.495,160.532
C06314=1020.820,425.071,338.672,174.426,50.497,160.535
C06315=1020.833,425.316,338.622,174.442,50.499,160.538
C06316=1020.845,425.560,338.573,174.457,50.500,160.541
C06317=1020.857,425.806,338.524,174.472,50.502,160.544
C06318=1020.869,426.050,338.474,174.488,50.504,160.548
C06319=1020.881,426.295,338.425,174.503,50.506,160.551
C06320=1020.893,426.540,338.375,174.518,50.508,160.554
C06321=1020.515,424.580,338.433,174.384,50.563,160.547
C06322=1020.503,424.334,338.482,174.368,50.562,160.543
C06323=1020.491,424.090,338.530,174.353,50.560,160.540
C06324=1020.479,423.844,338.580,174.338,50.558,160.537
C06325=1020.466,423.600,338.628,174.323,50.557,160.534
C06326=1020.455,423.354,338.677,174.307,50.555,160.531
C06327=1020.443,423.109,338.726,174.293,50.554,160.528
C06328=1020.431,422.865,338.774,174.278,50.552,160.525
C06329=1020.419,422.619,338.824,174.263,50.551,160.522
C06330=1020.407,422.374,338.871,174.248,50.550,160.519
C06331=1020.396,422.130,338.920,174.233,50.548,160.516
C06332=1020.384,421.885,338.969,174.219,50.547,160.513
C06333=1020.373,421.640,339.017,174.204,50.545,160.510
C06334=1020.360,421.395,339.066,174.190,50.544,160.507
C06335=1020.349,421.149,339.114,174.175,50.542,160.504
C06336=1020.337,420.904,339.162,174.160,50.541,160.501
C06337=1020.326,420.659,339.210,174.146,50.540,160.498
C06338=1020.314,420.414,339.259,174.131,50.539,160.495
C06339=1020.302,420.169,339.306,174.117,50.537,160.493
C06340=1020.291,419.924,339.355,174.102,50.536,160.489
C06341=1020.279,419.679,339.402,174.088,50.534,160.487
C06342=1020.268,419.434,339.451,174.074,50.533,160.484
C06343=1020.256,419.189,339.498,174.059,50.532,160.481
C06344=1020.244,418.943,339.546,174.045,50.531,160.478
C06345=1020.233,418.698,339.594,174.031,50.530,160.475
C06346=1020.222,418.452,339.641,174.017,50.528,160.473
C06347=1020.210,418.207,339.689,174.003,50.527,160.470
C06348=1020.199,417.962,339.737,173.988,50.526,160.467
C06349=1020.188,417.717,339.784,173.975,50.525,160.464
C06350=1020.176,417.472,339.832,173.960,50.524,160.461
C06351=1020.165,417.227,339.880,173.946,50.523,160.459
C06352=1020.153,416.981,339.927,173.933,50.522,160.456
C06353=1020.142,416.737,339.974,173.918,50.520,160.453
C06354=1020.131,416.491,340.022,173.905,50.519,160.451
C06355=1020.119,416.246,340.070,173.891,50.518,160.448
C06356=1020.108,416.001,340.116,173.878,50.517,160.445
C06357=1020.098,415.755,340.164,173.864,50.516,160.443
C06358=1020.086,415.510,340.211,173.850,50.515,160.440
C06359=1020.075,415.265,340.258,173.837,50.514,160.437
C06360=1020.065,415.019,340.305,173.823,50.513,160.435
C06361=1020.053,414.774,340.352,173.810,50.512,160.432
C06362=1020.042,414.529,340.399,173.795,50.511,160.429
C06363=1020.031,414.283,340.446,173.782,50.510,160.427
C06364=1020.020,414.038,340.493,173.769,50.509,160.424
C06365=1020.008,413.792,340.540,173.755,50.508,160.421
C06366=1019.997,413.547,340.586,173.742,50.507,160.419
C06367=1019.986,413.302,340.633,173.729,50.507,160.416
C06368=1019.976,413.056,340.680,173.715,50.506,160.414
C06369=1019.965,412.811,340.726,173.702,50.505,160.411
C06370=1019.953,412.544,340.776,173.687,50.504,160.408
C06371=1019.941,412.277,340.827,173.673,50.503,160.406
C06372=1019.929,412.011,340.877,173.659,50.502,160.403
C06373=1019.917,411.745,340.928,173.644,50.501,160.400
C06374=1019.907,411.498,340.975,173.632,50.501,160.398
C06375=1019.896,411.253,341.021,173.619,50.500,160.395
C06376=1019.885,411.008,341.067,173.606,50.499,160.393
C06377=1019.874,410.763,341.114,173.593,50.498,160.390
C06378=1019.864,410.517,341.160,173.580,50.498,160.388
C06379=1019.853,410.272,341.206,173.567,50.496,160.385
C06380=1019.842,410.026,341.251,173.554,50.496,160.383
C06381=1019.831,409.781,341.298,173.542,50.495,160.381
C06382=1019.821,409.536,341.344,173.528,50.494,160.378
C06383=1019.810,409.290,341.390,173.516,50.494,160.376
C06384=1019.800,409.044,341.436,173.503,50.493,160.374
C06385=1019.790,408.798,341.482,173.490,50.493,160.371
C06386=1019.778,408.553,341.528,173.478,50.492,160.369
C06387=1019.768,408.308,341.573,173.464,50.491,160.366
C06388=1019.758,408.062,341.618,173.452,50.491,160.364
C06389=1019.747,407.816,341.664,173.439,50.491,160.362
C06390=1019.736,407.571,341.710,173.427,50.490,160.359
C06391=1019.725,407.326,341.755,173.414,50.490,160.357
C06392=1019.715,407.079,341.801,173.402,50.489,160.355
C06393=1019.705,406.835,341.846,173.389,50.488,160.353
C06394=1019.694,406.589,341.891,173.377,50.488,160.350
C06395=1019.683,406.343,341.937,173.364,50.487,160.348
C06396=1019.673,406.097,341.982,173.353,50.487,160.346
C06397=1019.663,405.852,342.027,173.340,50.487,160.343
C06398=1019.652,405.606,342.072,173.327,50.486,160.341
C06399=1019.642,405.361,342.118,173.315,50.486,160.339
C06400=1019.632,405.115,342.163,173.303,50.485,160.337
C06401=1019.622,404.869,342.208,173.291,50.485,160.335
C06402=1019.612,404.623,342.253,173.278,50.485,160.332
C06403=1019.600,404.378,342.298,173.267,50.484,160.330
C06404=1019.591,404.132,342.343,173.254,50.484,160.328
C06405=1019.581,403.887,342.388,173.243,50.484,160.326
C06406=1019.571,403.641,342.433,173.230,50.484,160.324
C06407=1019.560,403.395,342.477,173.218,50.483,160.321
C06408=1019.550,403.149,342.522,173.206,50.483,160.319
C06409=1019.540,402.904,342.567,173.194,50.483,160.317
C06410=1019.530,402.658,342.612,173.182,50.482,160.315
C06411=1019.519,402.412,342.657,173.170,50.482,160.313
C06412=1019.510,402.167,342.701,173.159,50.482,160.311
C06413=1019.500,401.921,342.746,173.147,50.481,160.309
C06414=1019.490,401.676,342.791,173.135,50.481,160.307
C06415=1019.479,401.429,342.835,173.124,50.481,160.304
C06416=1019.470,401.184,342.880,173.111,50.481,160.302
C06417=1019.460,400.938,342.925,173.100,50.481,160.300
C06418=1019.451,400.692,342.969,173.088,50.481,160.298
C06419=1019.440,400.447,343.013,173.076,50.480,160.296
C06420=1019.431,400.201,343.057,173.065,50.480,160.294
C06421=1019.420,399.955,343.102,173.053,50.480,160.292
C06422=1019.410,399.709,343.146,173.041,50.480,160.290
C06423=1019.401,399.463,343.191,173.030,50.480,160.288
C06424=1019.390,399.217,343.234,173.018,50.480,160.286
C06425=1019.381,398.971,343.278,173.007,50.480,160.284
C06426=1019.371,398.726,343.323,172.996,50.480,160.282
C06427=1019.361,398.480,343.366,172.984,50.480,160.280
C06428=1019.352,398.234,343.411,172.972,50.480,160.278
C06429=1019.342,397.988,343.454,172.961,50.480,160.276
C06430=1019.329,397.658,343.513,172.946,50.479,160.273
C06431=1019.315,397.329,343.572,172.930,50.480,160.271
C06432=1019.303,397.000,343.630,172.916,50.480,160.268
C06433=1019.289,396.670,343.689,172.901,50.480,160.266
C06434=1019.280,396.424,343.733,172.890,50.480,160.264
C06435=1019.270,396.178,343.776,172.879,50.480,160.262
C06436=1019.260,395.933,343.820,172.867,50.481,160.260
C06437=1019.251,395.686,343.863,172.856,50.481,160.258
C06438=1019.241,395.441,343.906,172.845,50.481,160.256
C06439=1019.231,395.195,343.950,172.833,50.481,160.254
C06440=1019.222,394.948,343.993,172.822,50.481,160.252
C06441=1019.212,394.703,344.036,172.812,50.481,160.251
C06442=1019.202,394.457,344.079,172.801,50.481,160.249
C06443=1019.193,394.210,344.123,172.790,50.482,160.247
C06444=1019.184,393.965,344.166,172.779,50.482,160.245
C06445=1019.174,393.719,344.210,172.768,50.482,160.243
C06446=1019.165,393.473,344.252,172.757,50.482,160.241
C06447=1019.155,393.227,344.296,172.746,50.482,160.240
C06448=1019.146,392.980,344.339,172.735,50.483,160.238
C06449=1019.137,392.734,344.382,172.724,50.483,160.236
C06450=1019.127,392.489,344.425,172.713,50.484,160.234
C06451=1019.118,392.243,344.468,172.702,50.484,160.232
C06452=1019.108,391.996,344.511,172.692,50.484,160.231
C06453=1019.099,391.750,344.553,172.681,50.485,160.229
C06454=1019.089,391.504,344.596,172.670,50.485,160.227
C06455=1019.080,391.258,344.639,172.659,50.485,160.225
C06456=1019.071,391.011,344.682,172.650,50.486,160.224
C06457=1019.061,390.766,344.724,172.639,50.486,160.222
C06458=1019.052,390.519,344.767,172.628,50.487,160.220
C06459=1019.042,390.274,344.810,172.617,50.487,160.219
C06460=1019.033,390.028,344.852,172.607,50.488,160.217
C06461=1019.024,389.781,344.895,172.596,50.488,160.215
C06462=1019.015,389.535,344.938,172.586,50.488,160.214
C06463=1019.006,389.289,344.980,172.575,50.489,160.212
C06464=1018.997,389.043,345.022,172.564,50.489,160.210
C06465=1018.987,388.797,345.065,172.554,50.490,160.208
C06466=1018.979,388.550,345.107,172.544,50.490,160.207
C06467=1018.969,388.304,345.150,172.533,50.491,160.205
C06468=1018.960,388.059,345.192,172.523,50.492,160.203
C06469=1018.951,387.811,345.234,172.512,50.492,160.202
C06470=1018.941,387.566,345.276,172.503,50.493,160.200
C06471=1018.932,387.319,345.318,172.492,50.494,160.199
C06472=1018.924,387.073,345.360,172.481,50.494,160.197
C06473=1018.914,386.827,345.402,172.472,50.494,160.195
C06474=1018.905,386.581,345.444,172.461,50.495,160.194
C06475=1018.896,386.334,345.486,172.451,50.496,160.192
C06476=1018.887,386.088,345.529,172.441,50.496,160.191
C06477=1018.878,385.842,345.570,172.430,50.497,160.189
C06478=1018.869,385.595,345.612,172.420,50.498,160.187
C06479=1018.860,385.349,345.654,172.411,50.499,160.186
C06480=1018.851,385.103,345.696,172.400,50.500,160.184
C06481=1018.842,384.857,345.738,172.390,50.500,160.183
C06482=1018.833,384.610,345.779,172.380,50.501,160.181
C06483=1018.824,384.364,345.821,172.370,50.502,160.180
C06484=1018.814,384.117,345.862,172.360,50.503,160.178
C06485=1018.805,383.871,345.903,172.350,50.503,160.177
C06486=1018.796,383.625,345.945,172.341,50.504,160.175
C06487=1018.788,383.378,345.987,172.330,50.505,160.174
C06488=1018.778,383.132,346.028,172.319,50.506,160.172
C06489=1018.770,382.886,346.069,172.310,50.507,160.171
C06490=1018.759,382.595,346.119,172.299,50.508,160.169
C06491=1018.749,382.303,346.167,172.287,50.509,160.167
C06492=1018.738,382.011,346.216,172.275,50.510,160.165
C06493=1018.728,381.719,346.265,172.264,50.511,160.164
C06494=1018.719,381.472,346.306,172.254,50.512,160.162
C06495=1018.709,381.226,346.347,172.244,50.513,160.161
C06496=1018.701,380.980,346.388,172.234,50.514,160.159
C06497=1018.692,380.733,346.429,172.225,50.515,160.158
C06498=1018.684,380.486,346.470,172.214,50.517,160.157
C06499=1018.675,380.240,346.512,172.205,50.517,160.155
C06500=1018.666,379.994,346.552,172.196,50.518,160.154
C06501=1018.657,379.748,346.594,172.186,50.519,160.152
C06502=1018.648,379.501,346.635,172.176,50.520,160.151
C06503=1018.640,379.254,346.675,172.166,50.522,160.150
C06504=1018.631,379.008,346.717,172.157,50.522,160.148
C06505=1018.623,378.762,346.757,172.147,50.523,160.147
C06506=1018.614,378.515,346.798,172.137,50.525,160.145
C06507=1018.606,378.269,346.839,172.128,50.526,160.144
C06508=1018.597,378.022,346.880,172.119,50.527,160.143
C06509=1018.589,377.776,346.920,172.109,50.528,160.141
C06510=1018.580,377.529,346.962,172.100,50.529,160.140
C06511=1018.572,377.283,347.002,172.090,50.530,160.139
C06512=1018.563,377.036,347.043,172.080,50.531,160.137
C06513=1018.554,376.790,347.083,172.071,50.532,160.136
C06514=1018.546,376.543,347.124,172.062,50.533,160.135
C06515=1018.538,376.297,347.165,172.053,50.535,160.134
C06516=1018.530,376.051,347.206,172.043,50.536,160.132
C06517=1018.521,375.803,347.245,172.034,50.537,160.131
C06518=1018.513,375.557,347.286,172.025,50.538,160.130
C06519=1018.503,375.310,347.326,172.016,50.540,160.128
C06520=1018.495,375.064,347.367,172.006,50.541,160.127
C06521=1018.487,374.817,347.406,171.997,50.542,160.126
C06522=1018.478,374.570,347.447,171.988,50.544,160.125
C06523=1018.470,374.324,347.487,171.979,50.545,160.123
C06524=1018.462,374.078,347.527,171.970,50.547,160.122
C06525=1018.453,373.830,347.567,171.960,50.548,160.121
C06526=1018.444,373.584,347.607,171.951,50.550,160.120
C06527=1018.436,373.337,347.647,171.942,50.551,160.118
C06528=1018.427,373.091,347.687,171.933,50.552,160.117
C06529=1018.419,372.844,347.727,171.924,50.553,160.116
C06530=1018.410,372.598,347.767,171.914,50.555,160.115
C06531=1018.402,372.351,347.807,171.905,50.557,160.114
C06532=1018.394,372.104,347.846,171.896,50.558,160.112
C06533=1018.386,371.858,347.886,171.887,50.559,160.111
C06534=1018.378,371.611,347.926,171.878,50.561,160.110
C06535=1018.368,371.364,347.966,171.869,50.562,160.109
C06536=1018.361,371.117,348.006,171.860,50.564,160.108
C06537=1018.352,370.871,348.045,171.852,50.565,160.106
C06538=1018.345,370.624,348.085,171.842,50.567,160.105
C06539=1018.336,370.378,348.125,171.833,50.569,160.104
C06540=1018.327,370.131,348.165,171.824,50.570,160.103
C06541=1018.320,369.884,348.205,171.815,50.571,160.102
C06542=1018.311,369.638,348.244,171.806,50.573,160.101
C06543=1018.303,369.391,348.284,171.798,50.575,160.099
C06544=1018.295,369.144,348.323,171.789,50.576,160.098
C06545=1018.287,368.897,348.363,171.780,50.578,160.097
C06546=1018.279,368.651,348.402,171.771,50.579,160.096
C06547=1018.270,368.404,348.442,171.762,50.581,160.095
C06548=1018.263,368.157,348.482,171.754,50.583,160.094
C06549=1018.255,367.911,348.520,171.745,50.584,160.093
C06550=1018.247,367.641,348.564,171.735,50.586,160.092
C06551=1018.238,367.371,348.607,171.726,50.588,160.090
C06552=1018.228,367.102,348.649,171.716,50.590,160.089
C06553=1018.219,366.832,348.691,171.707,50.592,160.088
C06554=1018.211,366.586,348.731,171.698,50.593,160.087
C06555=1018.203,366.339,348.769,171.690,50.596,160.086
C06556=1018.195,366.092,348.809,171.681,50.597,160.085
C06557=1018.187,365.845,348.847,171.672,50.599,160.084
C06558=1018.179,365.598,348.887,171.664,50.601,160.083
C06559=1018.171,365.351,348.925,171.655,50.603,160.082
C06560=1018.163,365.105,348.964,171.646,50.604,160.081
C06561=1018.155,364.858,349.003,171.638,50.606,160.080
C06562=1018.147,364.611,349.042,171.629,50.608,160.079
C06563=1018.138,364.364,349.081,171.621,50.610,160.078
C06564=1018.131,364.118,349.119,171.613,50.611,160.077
C06565=1018.122,363.870,349.158,171.604,50.614,160.076
C06566=1018.115,363.623,349.197,171.595,50.615,160.075
C06567=1018.107,363.377,349.236,171.587,50.618,160.074
C06568=1018.099,363.130,349.274,171.579,50.620,160.073
C06569=1018.091,362.883,349.313,171.570,50.621,160.072
C06570=1018.083,362.636,349.351,171.561,50.624,160.071
C06571=1018.075,362.389,349.390,171.553,50.625,160.070
C06572=1018.068,362.142,349.428,171.545,50.627,160.069
C06573=1018.059,361.895,349.467,171.537,50.629,160.068
C06574=1018.052,361.649,349.505,171.528,50.631,160.067
C06575=1018.044,361.401,349.544,171.520,50.633,160.066
C06576=1018.036,361.155,349.582,171.511,50.635,160.065
C06577=1018.029,360.907,349.621,171.503,50.638,160.064
C06578=1018.021,360.661,349.659,171.495,50.639,160.063
C06579=1018.013,360.414,349.698,171.487,50.641,160.062
C06580=1018.006,360.167,349.736,171.478,50.643,160.061
C06581=1017.997,359.920,349.775,171.470,50.645,160.060
C06582=1017.990,359.673,349.813,171.461,50.648,160.059
C06583=1017.982,359.426,349.852,171.454,50.650,160.059
C06584=1017.974,359.179,349.889,171.446,50.652,160.058
C06585=1017.967,358.933,349.927,171.437,50.654,160.057
C06586=1017.959,358.685,349.966,171.429,50.656,160.056
C06587=1017.951,358.438,350.004,171.420,50.658,160.055
C06588=1017.943,358.191,350.042,171.413,50.660,160.054
C06589=1017.935,357.944,350.079,171.405,50.663,160.053
C06590=1017.928,357.698,350.117,171.396,50.665,160.052
C06591=1017.920,357.450,350.155,171.388,50.667,160.051
C06592=1017.912,357.203,350.193,171.381,50.669,160.051
C06593=1017.905,356.956,350.231,171.373,50.672,160.050
C06594=1017.896,356.709,350.269,171.364,50.674,160.049
C06595=1017.889,356.462,350.307,171.356,50.676,160.048
C06596=1017.882,356.215,350.344,171.348,50.678,160.047
C06597=1017.874,355.968,350.382,171.340,50.681,160.047
C06598=1017.866,355.721,350.420,171.332,50.683,160.046
C06599=1017.858,355.474,350.457,171.323,50.685,160.045
C06600=1017.851,355.227,350.495,171.316,50.688,160.044
C06601=1017.844,354.980,350.533,171.308,50.690,160.043
C06602=1017.836,354.733,350.570,171.300,50.693,160.043
C06603=1017.828,354.486,350.607,171.292,50.695,160.042
C06604=1017.821,354.238,350.645,171.284,50.697,160.041
C06605=1017.813,353.992,350.683,171.276,50.700,160.040
C06606=1017.806,353.745,350.721,171.268,50.702,160.039
C06607=1017.798,353.498,350.758,171.261,50.704,160.039
C06608=1017.791,353.251,350.795,171.252,50.707,160.038
C06609=1017.783,353.004,350.832,171.244,50.710,160.037
C06610=1017.775,352.741,350.872,171.236,50.712,160.036
C06611=1017.767,352.479,350.911,171.228,50.715,160.035
C06612=1017.759,352.218,350.951,171.220,50.717,160.035
C06613=1017.750,351.956,350.990,171.212,50.720,160.034
C06614=1017.743,351.709,351.028,171.204,50.722,160.033
C06615=1017.736,351.461,351.064,171.196,50.725,160.032
C06616=1017.728,351.214,351.101,171.189,50.728,160.032
C06617=1017.721,350.967,351.139,171.180,50.730,160.031
C06618=1017.713,350.720,351.176,171.173,50.733,160.030
C06619=1017.706,350.472,351.213,171.165,50.735,160.030
C06620=1017.698,350.226,351.250,171.157,50.738,160.029
C06621=1017.691,349.978,351.287,171.150,50.741,160.028
C06622=1017.683,349.731,351.323,171.142,50.743,160.027
C06623=1017.676,349.484,351.361,171.134,50.746,160.027
C06624=1017.669,349.237,351.398,171.127,50.748,160.026
C06625=1017.661,348.989,351.435,171.119,50.751,160.025
C06626=1017.654,348.743,351.472,171.112,50.754,160.025
C06627=1017.647,348.495,351.508,171.104,50.756,160.024
C06628=1017.640,348.248,351.545,171.096,50.759,160.023
C06629=1017.632,348.001,351.582,171.089,50.762,160.023
C06630=1017.625,347.754,351.619,171.081,50.765,160.022
C06631=1017.618,347.507,351.655,171.074,50.767,160.021
C06632=1017.610,347.260,351.693,171.066,50.770,160.021
C06633=1017.603,347.012,351.729,171.059,50.773,160.020
C06634=1017.596,346.765,351.766,171.051,50.775,160.019
C06635=1017.589,346.518,351.801,171.043,50.778,160.019
C06636=1017.581,346.271,351.838,171.036,50.781,160.018
C06637=1017.574,346.023,351.875,171.028,50.784,160.017
C06638=1017.566,345.776,351.911,171.021,50.787,160.017
C06639=1017.559,345.529,351.947,171.013,50.790,160.016
C06640=1017.552,345.281,351.984,171.006,50.792,160.015
C06641=1017.544,345.034,352.020,170.998,50.796,160.015
C06642=1017.537,344.787,352.056,170.990,50.798,160.014
C06643=1017.530,344.540,352.094,170.983,50.801,160.014
C06644=1017.522,344.293,352.130,170.976,50.804,160.013
C06645=1017.515,344.046,352.166,170.969,50.807,160.013
C06646=1017.508,343.798,352.202,170.961,50.810,160.012
C06647=1017.501,343.551,352.239,170.954,50.813,160.011
C06648=1017.494,343.304,352.275,170.946,50.816,160.011
C06649=1017.486,343.056,352.310,170.940,50.819,160.010
C06650=1017.480,342.809,352.347,170.932,50.822,160.010
C06651=1017.472,342.561,352.383,170.925,50.825,160.009
C06652=1017.465,342.315,352.419,170.917,50.828,160.008
C06653=1017.457,342.067,352.455,170.910,50.831,160.008
C06654=1017.451,341.820,352.491,170.902,50.834,160.007
C06655=1017.444,341.572,352.527,170.896,50.837,160.007
C06656=1017.437,341.325,352.563,170.888,50.840,160.006
C06657=1017.429,341.078,352.599,170.881,50.843,160.006
C06658=1017.423,340.831,352.635,170.873,50.846,160.005
C06659=1017.415,340.583,352.671,170.866,50.849,160.005
C06660=1017.408,340.336,352.707,170.859,50.852,160.004
C06661=1017.400,340.088,352.743,170.852,50.855,160.004
C06662=1017.394,339.841,352.778,170.844,50.858,160.003
C06663=1017.387,339.594,352.814,170.838,50.861,160.003
C06664=1017.380,339.346,352.850,170.830,50.865,160.002
C06665=1017.373,339.099,352.886,170.823,50.867,160.001
C06666=1017.366,338.851,352.921,170.815,50.871,160.001
C06667=1017.359,338.604,352.957,170.809,50.874,160.001
C06668=1017.352,338.357,352.992,170.801,50.877,160.000
C06669=1017.344,338.110,353.029,170.794,50.881,160.000
C06670=1017.336,337.845,353.066,170.787,50.884,159.999
C06671=1017.329,337.580,353.104,170.779,50.888,159.999
C06672=1017.322,337.316,353.142,170.772,50.891,159.998
C06673=1017.314,337.051,353.180,170.764,50.895,159.998
C06674=1017.307,336.804,353.215,170.756,50.898,159.997
C06675=1017.300,336.555,353.250,170.750,50.901,159.997
C06676=1017.293,336.309,353.286,170.743,50.904,159.996
C06677=1017.286,336.061,353.321,170.736,50.908,159.996
C06678=1017.279,335.814,353.356,170.729,50.911,159.995
C06679=1017.272,335.566,353.392,170.721,50.914,159.995
C06680=1017.265,335.319,353.427,170.715,50.918,159.994
C06681=1017.258,335.071,353.462,170.707,50.921,159.994
C06682=1017.252,334.824,353.497,170.701,50.924,159.994
C06683=1017.245,334.576,353.532,170.693,50.928,159.993
C06684=1017.237,334.328,353.568,170.687,50.932,159.993
C06685=1017.231,334.081,353.603,170.680,50.935,159.992
C06686=1017.224,333.834,353.639,170.672,50.938,159.992
C06687=1017.216,333.587,353.673,170.666,50.941,159.991
C06688=1017.210,333.339,353.708,170.659,50.945,159.991
C06689=1017.203,333.092,353.743,170.652,50.949,159.991
C06690=1017.196,332.845,353.778,170.645,50.952,159.990
C06691=1017.189,332.597,353.813,170.638,50.955,159.990
C06692=1017.183,332.350,353.848,170.632,50.959,159.990
C06693=1017.176,332.102,353.884,170.624,50.963,159.989
C06694=1017.168,331.855,353.918,170.618,50.966,159.989
C06695=1017.161,331.607,353.953,170.610,50.970,159.988
C06696=1017.154,331.359,353.988,170.604,50.973,159.988
C06697=1017.148,331.112,354.023,170.597,50.977,159.988
C06698=1017.141,330.864,354.057,170.590,50.980,159.987
C06699=1017.134,330.617,354.092,170.583,50.984,159.987
C06700=1017.127,330.370,354.127,170.576,50.988,159.987
C06701=1017.120,330.122,354.161,170.570,50.991,159.986
C06702=1017.113,329.874,354.196,170.563,50.995,159.986
C06703=1017.107,329.627,354.230,170.556,50.999,159.986
C06704=1017.100,329.380,354.265,170.550,51.002,159.985
C06705=1017.093,329.132,354.299,170.542,51.006,159.985
C06706=1017.086,328.885,354.334,170.536,51.010,159.985
C06707=1017.079,328.637,354.368,170.529,51.013,159.984
C06708=1017.072,328.390,354.403,170.522,51.017,159.984
C06709=1017.066,328.142,354.438,170.516,51.021,159.984
C06710=1017.059,327.894,354.473,170.508,51.024,159.983
C06711=1017.052,327.647,354.507,170.502,51.028,159.983
C06712=1017.046,327.399,354.541,170.496,51.032,159.983
C06713=1017.039,327.152,354.576,170.488,51.036,159.983
C06714=1017.032,326.904,354.610,170.482,51.039,159.982
C06715=1017.026,326.656,354.644,170.476,51.043,159.982
C06716=1017.019,326.409,354.679,170.468,51.047,159.982
C06717=1017.012,326.162,354.713,170.462,51.051,159.981
C06718=1017.006,325.914,354.747,170.455,51.055,159.981
C06719=1016.999,325.666,354.781,170.448,51.058,159.981
C06720=1016.991,325.419,354.815,170.442,51.062,159.980
C06721=1016.985,325.172,354.848,170.435,51.066,159.980
C06722=1016.978,324.924,354.882,170.429,51.070,159.980
C06723=1016.971,324.676,354.917,170.422,51.075,159.980
C06724=1016.964,324.428,354.950,170.416,51.079,159.980
C06725=1016.957,324.181,354.984,170.409,51.083,159.979
C06726=1016.950,323.934,355.018,170.402,51.087,159.979
C06727=1016.944,323.686,355.052,170.396,51.090,159.979
C06728=1016.937,323.438,355.086,170.389,51.095,159.979
C06729=1016.930,323.191,355.119,170.383,51.098,159.978
C06730=1016.922,322.921,355.156,170.375,51.103,159.978
C06731=1016.915,322.653,355.193,170.369,51.107,159.978
C06732=1016.908,322.384,355.229,170.361,51.112,159.978
C06733=1016.901,322.115,355.265,170.355,51.116,159.978
C06734=1016.894,321.867,355.299,170.347,51.120,159.977
C06735=1016.887,321.619,355.333,170.341,51.124,159.977
C06736=1016.880,321.372,355.367,170.334,51.128,159.977
C06737=1016.874,321.124,355.400,170.328,51.132,159.977
C06738=1016.867,320.877,355.433,170.322,51.137,159.977
C06739=1016.861,320.629,355.468,170.315,51.141,159.976
C06740=1016.854,320.381,355.501,170.309,51.145,159.976
C06741=1016.847,320.134,355.534,170.302,51.150,159.976
C06742=1016.840,319.886,355.568,170.296,51.153,159.976
C06743=1016.834,319.638,355.602,170.289,51.157,159.975
C06744=1016.827,319.391,355.635,170.283,51.162,159.975
C06745=1016.821,319.143,355.668,170.276,51.166,159.975
C06746=1016.814,318.895,355.702,170.271,51.170,159.975
C06747=1016.807,318.648,355.735,170.263,51.174,159.975
C06748=1016.801,318.400,355.769,170.257,51.178,159.975
C06749=1016.794,318.153,355.803,170.251,51.183,159.975
C06750=1016.788,317.905,355.835,170.244,51.187,159.974
C06751=1016.781,317.657,355.869,170.238,51.191,159.974
C06752=1016.775,317.410,355.903,170.232,51.195,159.974
C06753=1016.768,317.161,355.936,170.225,51.200,159.974
C06754=1016.762,316.914,355.969,170.219,51.204,159.974
C06755=1016.755,316.667,356.002,170.212,51.209,159.974
C06756=1016.748,316.419,356.036,170.206,51.212,159.973
C06757=1016.743,316.171,356.069,170.200,51.217,159.973
C06758=1016.736,315.924,356.102,170.193,51.222,159.973
C06759=1016.729,315.676,356.136,170.187,51.226,159.973
C06760=1016.723,315.428,356.168,170.181,51.230,159.973
C06761=1016.717,315.181,356.201,170.174,51.234,159.973
C06762=1016.711,314.933,356.234,170.168,51.239,159.973
C06763=1016.704,314.685,356.268,170.163,51.243,159.973
C06764=1016.698,314.437,356.301,170.156,51.247,159.973
C06765=1016.691,314.190,356.334,170.150,51.252,159.972
C06766=1016.685,313.942,356.366,170.144,51.256,159.972
C06767=1016.678,313.694,356.401,170.138,51.261,159.972
C06768=1016.672,313.447,356.434,170.131,51.265,159.972
C06769=1016.666,313.199,356.466,170.125,51.269,159.972
C06770=1016.660,312.952,356.499,170.119,51.274,159.972
C06771=1016.653,312.704,356.532,170.112,51.279,159.972
C06772=1016.647,312.455,356.566,170.107,51.283,159.972
C06773=1016.641,312.208,356.598,170.100,51.287,159.972
C06774=1016.634,311.961,356.632,170.094,51.292,159.972
C06775=1016.628,311.713,356.664,170.088,51.296,159.972
C06776=1016.622,311.466,356.697,170.082,51.301,159.972
C06777=1016.616,311.218,356.731,170.076,51.305,159.972
C06778=1016.610,310.970,356.763,170.069,51.310,159.972
C06779=1016.604,310.723,356.796,170.064,51.315,159.971
C06780=1016.597,310.475,356.829,170.057,51.318,159.971
C06781=1016.591,310.227,356.862,170.051,51.323,159.971
C06782=1016.585,309.979,356.895,170.045,51.328,159.971
C06783=1016.579,309.731,356.927,170.039,51.332,159.971
C06784=1016.573,309.484,356.960,170.033,51.337,159.971
C06785=1016.566,309.236,356.992,170.027,51.342,159.971
C06786=1016.559,308.988,357.025,170.021,51.347,159.971
C06787=1016.553,308.740,357.057,170.014,51.352,159.971
C06788=1016.546,308.493,357.089,170.008,51.356,159.971
C06789=1016.540,308.244,357.121,170.003,51.361,159.971
C06790=1016.533,307.981,357.155,169.996,51.366,159.971
C06791=1016.527,307.718,357.190,169.990,51.372,159.971
C06792=1016.519,307.454,357.224,169.983,51.376,159.971
C06793=1016.512,307.190,357.257,169.977,51.382,159.971
C06794=1016.506,306.942,357.290,169.971,51.386,159.971
C06795=1016.500,306.695,357.322,169.964,51.391,159.971
C06796=1016.493,306.447,357.354,169.959,51.396,159.971
C06797=1016.487,306.199,357.386,169.952,51.401,159.971
C06798=1016.480,305.951,357.418,169.946,51.406,159.971
C06799=1016.474,305.703,357.450,169.941,51.411,159.971
C06800=1016.467,305.456,357.482,169.934,51.416,159.971
C06801=1016.462,305.208,357.514,169.928,51.421,159.972
C06802=1016.455,304.960,357.545,169.922,51.426,159.971
C06803=1016.449,304.713,357.578,169.916,51.431,159.972
C06804=1016.443,304.465,357.610,169.910,51.435,159.972
C06805=1016.436,304.217,357.641,169.904,51.441,159.972
C06806=1016.430,303.968,357.673,169.898,51.445,159.972
C06807=1016.423,303.721,357.706,169.893,51.451,159.972
C06808=1016.417,303.473,357.738,169.886,51.455,159.972
C06809=1016.410,303.225,357.769,169.881,51.461,159.972
C06810=1016.405,302.978,357.801,169.874,51.466,159.972
C06811=1016.398,302.730,357.832,169.869,51.471,159.972
C06812=1016.392,302.482,357.865,169.863,51.476,159.972
C06813=1016.385,302.234,357.896,169.856,51.481,159.972
C06814=1016.379,301.986,357.928,169.851,51.486,159.972
C06815=1016.374,301.738,357.960,169.845,51.491,159.972
C06816=1016.367,301.491,357.991,169.839,51.496,159.972
C06817=1016.361,301.242,358.023,169.833,51.501,159.973
C06818=1016.354,300.994,358.055,169.827,51.507,159.973
C06819=1016.349,300.747,358.086,169.822,51.512,159.973
C06820=1016.342,300.499,358.118,169.816,51.516,159.973
C06821=1016.336,300.251,358.150,169.810,51.522,159.973
C06822=1016.329,300.003,358.181,169.804,51.527,159.973
C06823=1016.324,299.755,358.213,169.799,51.532,159.973
C06824=1016.317,299.507,358.244,169.792,51.537,159.973
C06825=1016.311,299.259,358.276,169.787,51.542,159.973
C06826=1016.306,299.012,358.308,169.780,51.548,159.973
C06827=1016.299,298.764,358.340,169.775,51.553,159.974
C06828=1016.293,298.516,358.372,169.769,51.558,159.974
C06829=1016.287,298.268,358.403,169.763,51.563,159.974
C06830=1016.281,298.020,358.434,169.757,51.568,159.974
C06831=1016.275,297.772,358.465,169.752,51.573,159.974
C06832=1016.269,297.524,358.497,169.746,51.579,159.974
C06833=1016.262,297.276,358.529,169.740,51.584,159.974
C06834=1016.257,297.029,358.560,169.735,51.589,159.975
C06835=1016.251,296.780,358.591,169.728,51.595,159.975
C06836=1016.245,296.533,358.623,169.723,51.600,159.975
C06837=1016.239,296.285,358.654,169.718,51.605,159.975
C06838=1016.233,296.037,358.686,169.711,51.611,159.975
C06839=1016.227,295.788,358.717,169.706,51.616,159.975
C06840=1016.221,295.541,358.748,169.700,51.621,159.975
C06841=1016.215,295.293,358.780,169.694,51.627,159.976
C06842=1016.209,295.045,358.811,169.689,51.632,159.976
C06843=1016.204,294.797,358.842,169.682,51.637,159.976
C06844=1016.197,294.549,358.874,169.677,51.642,159.976
C06845=1016.192,294.301,358.905,169.672,51.648,159.976
C06846=1016.185,294.054,358.937,169.665,51.653,159.976
C06847=1016.180,293.808,358.967,169.660,51.658,159.977
C06848=1016.174,293.561,358.998,169.655,51.664,159.977
C06849=1016.168,293.314,359.029,169.648,51.669,159.977
C06850=1016.162,293.067,359.060,169.643,51.675,159.977
C06851=1016.156,292.820,359.091,169.638,51.680,159.977
C06852=1016.150,292.573,359.122,169.632,51.686,159.978
C06853=1016.144,292.326,359.153,169.626,51.691,159.978
C06854=1016.138,292.079,359.184,169.621,51.697,159.978
C06855=1016.132,291.831,359.214,169.615,51.702,159.978
C06856=1016.126,291.583,359.245,169.610,51.708,159.978
C06857=1016.121,291.335,359.277,169.604,51.714,159.979
C06858=1016.114,291.087,359.307,169.598,51.719,159.979
C06859=1016.108,290.839,359.338,169.593,51.724,159.979
C06860=1016.102,290.591,359.368,169.587,51.730,159.979
C06861=1016.096,290.343,359.400,169.582,51.736,159.980
C06862=1016.090,290.095,359.430,169.576,51.742,159.980
C06863=1016.084,289.847,359.461,169.570,51.747,159.980
C06864=1016.078,289.599,359.491,169.564,51.753,159.980
C06865=1016.072,289.351,359.521,169.559,51.759,159.981
C06866=1016.065,289.103,359.552,169.553,51.765,159.981
C06867=1016.060,288.855,359.582,169.548,51.771,159.981
C06868=1016.054,288.607,359.613,169.542,51.776,159.981
C06869=1016.047,288.358,359.643,169.537,51.782,159.982
C06870=1016.042,288.111,359.674,169.531,51.787,159.982
C06871=1016.036,287.862,359.705,169.525,51.794,159.982
C06872=1016.031,287.615,359.735,169.520,51.799,159.983
C06873=1016.024,287.366,359.766,169.514,51.805,159.983
C06874=1016.018,287.118,359.796,169.509,51.811,159.983
C06875=1016.013,286.870,359.827,169.503,51.816,159.983
C06876=1016.006,286.622,359.857,169.498,51.822,159.984
C06877=1016.000,286.374,359.888,169.492,51.829,159.984
C06878=1015.994,286.127,359.917,169.487,51.834,159.984
C06879=1015.988,285.879,359.948,169.481,51.840,159.984
C06880=1015.982,285.631,359.978,169.476,51.846,159.985
C06881=1015.976,285.382,360.008,169.470,51.852,159.985
C06882=1015.970,285.134,360.038,169.465,51.858,159.985
C06883=1015.964,284.886,360.069,169.460,51.864,159.986
C06884=1015.959,284.638,360.099,169.454,51.870,159.986
C06885=1015.953,284.390,360.129,169.449,51.875,159.986
C06886=1015.947,284.141,360.159,169.443,51.882,159.987
C06887=1015.941,283.894,360.190,169.438,51.888,159.987
C06888=1015.935,283.645,360.219,169.432,51.894,159.987
C06889=1015.929,283.398,360.249,169.426,51.900,159.988
C06890=1015.923,283.150,360.280,169.421,51.906,159.988
C06891=1015.917,282.901,360.309,169.415,51.912,159.988
C06892=1015.910,282.653,360.339,169.410,51.918,159.989
C06893=1015.905,282.405,360.369,169.404,51.924,159.989
C06894=1015.899,282.157,360.399,169.399,51.930,159.989
C06895=1015.893,281.908,360.429,169.393,51.937,159.990
C06896=1015.887,281.661,360.459,169.388,51.943,159.990
C06897=1015.881,281.412,360.488,169.382,51.949,159.990
C06898=1015.876,281.165,360.519,169.378,51.955,159.991
C06899=1015.869,280.917,360.548,169.372,51.961,159.991
C06900=1015.864,280.669,360.578,169.367,51.968,159.992
C06901=1015.858,280.420,360.608,169.361,51.974,159.992
C06902=1015.852,280.172,360.638,169.356,51.980,159.992
C06903=1015.845,279.924,360.667,169.350,51.986,159.993
C06904=1015.840,279.675,360.697,169.345,51.992,159.993
C06905=1015.834,279.427,360.727,169.340,51.998,159.993
C06906=1015.829,279.187,360.756,169.335,52.004,159.994
C06907=1015.823,278.946,360.784,169.329,52.010,159.994
C06908=1015.818,278.706,360.814,169.324,52.017,159.995
C06909=1015.812,278.464,360.843,169.319,52.023,159.995
C06910=1015.806,278.224,360.871,169.313,52.029,159.995
C06911=1015.801,277.984,360.900,169.308,52.035,159.996
C06912=1015.795,277.743,360.929,169.304,52.041,159.996
C06913=1015.790,277.502,360.957,169.299,52.047,159.996
C06914=1015.784,277.254,360.986,169.293,52.053,159.997
C06915=1015.778,277.006,361.017,169.287,52.060,159.997
C06916=1015.772,276.758,361.046,169.282,52.066,159.998
C06917=1015.766,276.510,361.075,169.276,52.072,159.998
C06918=1015.761,276.261,361.105,169.272,52.079,159.999
C06919=1015.755,276.013,361.135,169.266,52.085,159.999
C06920=1015.749,275.765,361.164,169.261,52.092,159.999
C06921=1015.743,275.517,361.194,169.256,52.098,160.000
C06922=1015.737,275.269,361.223,169.250,52.105,160.000
C06923=1015.732,275.021,361.252,169.245,52.111,160.001
C06924=1015.726,274.773,361.281,169.240,52.118,160.001
C06925=1015.720,274.524,361.311,169.235,52.124,160.002
C06926=1015.714,274.276,361.340,169.229,52.131,160.002
C06927=1015.708,274.028,361.369,169.223,52.137,160.002
C06928=1015.702,273.779,361.398,169.219,52.144,160.003
C06929=1015.696,273.531,361.427,169.213,52.151,160.004
C06930=1015.691,273.282,361.457,169.209,52.157,160.004
C06931=1015.685,273.035,361.485,169.203,52.164,160.004
C06932=1015.679,272.787,361.515,169.197,52.170,160.005
C06933=1015.673,272.538,361.544,169.193,52.177,160.005
C06934=1015.668,272.290,361.574,169.187,52.184,160.006
C06935=1015.661,272.042,361.603,169.181,52.190,160.006
C06936=1015.657,271.794,361.631,169.177,52.197,160.007
C06937=1015.651,271.545,361.660,169.171,52.203,160.007
C06938=1015.644,271.297,361.689,169.166,52.210,160.008
C06939=1015.639,271.049,361.719,169.161,52.216,160.008
C06940=1015.633,270.801,361.748,169.156,52.223,160.009
C06941=1015.627,270.553,361.776,169.151,52.230,160.009
C06942=1015.622,270.304,361.806,169.146,52.237,160.010
C06943=1015.615,270.056,361.835,169.140,52.244,160.010
C06944=1015.611,269.808,361.863,169.135,52.250,160.011
C06945=1015.605,269.560,361.892,169.130,52.257,160.011
C06946=1015.598,269.311,361.921,169.124,52.264,160.012
C06947=1015.594,269.063,361.950,169.120,52.271,160.012
C06948=1015.588,268.815,361.979,169.114,52.278,160.013
C06949=1015.582,268.566,362.007,169.109,52.285,160.013
C06950=1015.576,268.319,362.036,169.104,52.291,160.014
C06951=1015.570,268.070,362.066,169.099,52.298,160.014
C06952=1015.564,267.822,362.094,169.094,52.305,160.015
C06953=1015.559,267.574,362.123,169.088,52.312,160.015
C06954=1015.553,267.325,362.151,169.084,52.319,160.016
C06955=1015.548,267.076,362.180,169.078,52.326,160.016
C06956=1015.542,266.829,362.208,169.073,52.333,160.017
C06957=1015.536,266.580,362.237,169.068,52.340,160.018
C06958=1015.530,266.332,362.266,169.063,52.347,160.018
C06959=1015.524,266.084,362.294,169.057,52.354,160.019
C06960=1015.519,265.836,362.323,169.052,52.361,160.019
C06961=1015.514,265.587,362.351,169.047,52.367,160.020
C06962=1015.508,265.339,362.380,169.042,52.374,160.020
C06963=1015.501,265.091,362.409,169.037,52.382,160.021
C06964=1015.496,264.843,362.437,169.031,52.389,160.021
C06965=1015.490,264.594,362.465,169.027,52.396,160.022
C06966=1015.485,264.355,362.493,169.022,52.403,160.023
C06967=1015.479,264.117,362.520,169.017,52.409,160.023
C06968=1015.474,263.878,362.547,169.012,52.416,160.024
C06969=1015.468,263.640,362.574,169.007,52.423,160.024
C06970=1015.463,263.402,362.601,169.002,52.430,160.025
C06971=1015.458,263.163,362.629,168.997,52.437,160.025
C06972=1015.452,262.925,362.656,168.992,52.444,160.026
C06973=1015.447,262.686,362.683,168.987,52.450,160.026
C06974=1015.441,262.438,362.711,168.982,52.458,160.027
C06975=1015.435,262.190,362.740,168.977,52.465,160.028
C06976=1015.430,261.941,362.768,168.973,52.472,160.028
C06977=1015.424,261.693,362.796,168.968,52.479,160.029
C06978=1015.419,261.445,362.824,168.962,52.486,160.030
C06979=1015.413,261.196,362.853,168.957,52.494,160.030
C06980=1015.407,260.948,362.881,168.952,52.501,160.031
C06981=1015.402,260.700,362.908,168.947,52.508,160.031
C06982=1015.396,260.451,362.937,168.942,52.516,160.032
C06983=1015.391,260.203,362.965,168.937,52.523,160.033
C06984=1015.385,259.954,362.993,168.932,52.530,160.033
C06985=1015.379,259.706,363.021,168.926,52.537,160.034
C06986=1015.373,259.457,363.049,168.921,52.545,160.034
C06987=1015.368,259.209,363.077,168.916,52.553,160.035
C06988=1015.362,258.962,363.105,168.912,52.560,160.036
C06989=1015.356,258.713,363.133,168.907,52.567,160.037
C06990=1015.350,258.465,363.160,168.902,52.575,160.037
C06991=1015.345,258.217,363.188,168.897,52.583,160.038
C06992=1015.339,257.968,363.216,168.892,52.590,160.038
C06993=1015.333,257.720,363.243,168.887,52.598,160.039
C06994=1015.327,257.471,363.271,168.882,52.605,160.040
C06995=1015.321,257.223,363.298,168.877,52.613,160.041
C06996=1015.316,256.975,363.326,168.871,52.620,160.041
C06997=1015.310,256.725,363.354,168.866,52.628,160.042
C06998=1015.304,256.478,363.381,168.861,52.636,160.043
C06999=1015.298,256.228,363.409,168.856,52.643,160.043
C07000=1015.292,255.981,363.436,168.851,52.651,160.044
C07001=1015.287,255.733,363.464,168.846,52.659,160.045
C07002=1015.281,255.483,363.492,168.841,52.667,160.045
C07003=1015.275,255.235,363.519,168.836,52.674,160.046
C07004=1015.270,254.987,363.546,168.831,52.681,160.047
C07005=1015.264,254.738,363.575,168.826,52.689,160.047
C07006=1015.258,254.490,363.602,168.821,52.697,160.048
C07007=1015.253,254.242,363.629,168.816,52.705,160.049
C07008=1015.247,253.994,363.657,168.811,52.712,160.050
C07009=1015.242,253.745,363.684,168.806,52.720,160.050
C07010=1015.236,253.496,363.712,168.801,52.728,160.051
C07011=1015.230,253.248,363.739,168.796,52.736,160.052
C07012=1015.225,252.999,363.766,168.791,52.743,160.052
C07013=1015.219,252.751,363.794,168.786,52.751,160.053
C07014=1015.214,252.502,363.821,168.781,52.759,160.054
C07015=1015.208,252.254,363.849,168.776,52.767,160.055
C07016=1015.203,252.006,363.876,168.771,52.774,160.055
C07017=1015.197,251.757,363.904,168.766,52.782,160.056
C07018=1015.191,251.509,363.931,168.761,52.790,160.057
C07019=1015.186,251.260,363.958,168.757,52.798,160.058
C07020=1015.180,251.012,363.986,168.752,52.806,160.058
C07021=1015.175,250.764,364.013,168.747,52.814,160.059
C07022=1015.169,250.514,364.040,168.742,52.822,160.060
C07023=1015.163,250.267,364.068,168.737,52.830,160.061
C07024=1015.158,250.018,364.095,168.732,52.837,160.061
C07025=1015.153,249.769,364.122,168.727,52.845,160.062
C07026=1015.147,249.531,364.149,168.722,52.853,160.063
C07027=1015.142,249.291,364.174,168.718,52.860,160.064
C07028=1015.137,249.051,364.201,168.713,52.868,160.064
C07029=1015.131,248.812,364.227,168.708,52.876,160.065
C07030=1015.126,248.572,364.253,168.705,52.883,160.066
C07031=1015.120,248.334,364.280,168.700,52.891,160.067
C07032=1015.116,248.094,364.306,168.695,52.899,160.067
C07033=1015.110,247.855,364.332,168.690,52.907,160.068
C07034=1015.105,247.606,364.359,168.685,52.915,160.069
C07035=1015.099,247.357,364.386,168.680,52.923,160.070
C07036=1015.094,247.108,364.413,168.675,52.931,160.070
C07037=1015.088,246.861,364.441,168.671,52.939,160.071
C07038=1015.083,246.612,364.468,168.666,52.947,160.072
C07039=1015.078,246.363,364.495,168.661,52.955,160.073
C07040=1015.072,246.115,364.522,168.657,52.963,160.074
C07041=1015.067,245.866,364.549,168.652,52.971,160.074
C07042=1015.061,245.618,364.576,168.647,52.979,160.075
C07043=1015.056,245.369,364.603,168.642,52.987,160.076
C07044=1015.051,245.121,364.630,168.636,52.996,160.077
C07045=1015.045,244.872,364.657,168.632,53.004,160.078
C07046=1015.040,244.624,364.684,168.627,53.012,160.078
C07047=1015.034,244.376,364.712,168.622,53.020,160.079
C07048=1015.029,244.127,364.739,168.617,53.028,160.080
C07049=1015.023,243.879,364.765,168.613,53.037,160.081
C07050=1015.018,243.630,364.793,168.608,53.045,160.082
C07051=1015.014,243.382,364.820,168.604,53.053,160.083
C07052=1015.008,243.134,364.846,168.599,53.061,160.083
C07053=1015.003,242.885,364.873,168.594,53.069,160.084
C07054=1014.997,242.637,364.900,168.588,53.078,160.085
C07055=1014.993,242.388,364.927,168.584,53.086,160.086
C07056=1014.987,242.139,364.953,168.579,53.095,160.087
C07057=1014.981,241.891,364.980,168.574,53.102,160.087
C07058=1014.975,241.642,365.007,168.570,53.111,160.088
C07059=1014.970,241.394,365.034,168.565,53.120,160.089
C07060=1014.965,241.145,365.060,168.560,53.128,160.090
C07061=1014.960,240.897,365.086,168.555,53.136,160.091
C07062=1014.955,240.648,365.113,168.551,53.145,160.092
C07063=1014.949,240.400,365.140,168.545,53.154,160.093
C07064=1014.943,240.151,365.166,168.541,53.162,160.094
C07065=1014.938,239.903,365.193,168.536,53.170,160.094
C07066=1014.933,239.654,365.220,168.532,53.179,160.095
C07067=1014.927,239.405,365.246,168.526,53.187,160.096
C07068=1014.922,239.157,365.272,168.522,53.196,160.097
C07069=1014.917,238.909,365.299,168.517,53.204,160.098
C07070=1014.911,238.660,365.325,168.513,53.213,160.099
C07071=1014.906,238.411,365.352,168.507,53.222,160.100
C07072=1014.900,238.163,365.378,168.503,53.230,160.101
C07073=1014.895,237.915,365.404,168.498,53.239,160.102
C07074=1014.889,237.666,365.431,168.493,53.248,160.102
C07075=1014.884,237.417,365.457,168.489,53.256,160.103
C07076=1014.878,237.169,365.483,168.484,53.265,160.104
C07077=1014.873,236.920,365.509,168.479,53.274,160.105
C07078=1014.868,236.672,365.535,168.474,53.282,160.106
C07079=1014.862,236.424,365.561,168.470,53.291,160.107
C07080=1014.856,236.175,365.587,168.464,53.300,160.108
C07081=1014.851,235.926,365.614,168.460,53.309,160.109
C07082=1014.845,235.677,365.640,168.455,53.317,160.110
C07083=1014.840,235.429,365.665,168.451,53.327,160.111
C07084=1014.835,235.181,365.692,168.446,53.335,160.112
C07085=1014.829,234.932,365.718,168.441,53.344,160.113
C07086=1014.824,234.689,365.744,168.436,53.353,160.114
C07087=1014.819,234.446,365.769,168.432,53.361,160.115
C07088=1014.814,234.203,365.794,168.428,53.370,160.116
C07089=1014.808,233.960,365.820,168.422,53.379,160.116
C07090=1014.803,233.718,365.845,168.418,53.387,160.117
C07091=1014.797,233.475,365.871,168.413,53.396,160.118
C07092=1014.792,233.232,365.896,168.409,53.405,160.119
C07093=1014.787,232.989,365.921,168.404,53.414,160.120
C07094=1014.782,232.741,365.947,168.400,53.423,160.121
C07095=1014.776,232.492,365.973,168.395,53.431,160.122
C07096=1014.771,232.243,365.999,168.390,53.441,160.123
C07097=1014.766,231.994,366.025,168.386,53.450,160.124
C07098=1014.760,231.745,366.051,168.380,53.459,160.125
C07099=1014.755,231.498,366.077,168.377,53.468,160.126
C07100=1014.750,231.249,366.103,168.371,53.477,160.127
C07101=1014.745,231.001,366.129,168.367,53.485,160.128
C07102=1014.739,230.752,366.155,168.362,53.495,160.129
C07103=1014.733,230.503,366.180,168.357,53.504,160.130
C07104=1014.728,230.255,366.205,168.352,53.513,160.131
C07105=1014.723,230.006,366.231,168.348,53.522,160.132
C07106=1014.717,229.757,366.257,168.343,53.532,160.133
C07107=1014.712,229.509,366.284,168.339,53.540,160.134
C07108=1014.707,229.260,366.310,168.334,53.550,160.135
C07109=1014.702,229.012,366.335,168.330,53.558,160.136
C07110=1014.696,228.763,366.361,168.325,53.568,160.137
C07111=1014.691,228.515,366.386,168.320,53.577,160.138
C07112=1014.686,228.265,366.411,168.315,53.586,160.139
C07113=1014.681,228.017,366.437,168.311,53.595,160.140
C07114=1014.675,227.768,366.463,168.306,53.605,160.141
C07115=1014.670,227.519,366.489,168.301,53.614,160.142
C07116=1014.664,227.271,366.514,168.297,53.623,160.143
C07117=1014.659,227.022,366.540,168.292,53.633,160.144
C07118=1014.654,226.774,366.565,168.288,53.642,160.145
C07119=1014.648,226.525,366.591,168.283,53.651,160.146
C07120=1014.643,226.277,366.616,168.278,53.661,160.147
C07121=1014.638,226.027,366.641,168.274,53.670,160.148
C07122=1014.633,225.779,366.667,168.269,53.680,160.149
C07123=1014.626,225.530,366.692,168.264,53.689,160.150
C07124=1014.622,225.282,366.718,168.260,53.698,160.151
C07125=1014.616,225.033,366.742,168.255,53.708,160.152
C07126=1014.611,224.784,366.768,168.250,53.717,160.154
C07127=1014.605,224.536,366.793,168.246,53.727,160.155
C07128=1014.600,224.287,366.818,168.241,53.736,160.156
C07129=1014.594,224.038,366.843,168.236,53.746,160.157
C07130=1014.589,223.790,366.869,168.232,53.756,160.158
C07131=1014.584,223.541,366.894,168.228,53.765,160.159
C07132=1014.578,223.292,366.919,168.223,53.775,160.160
C07133=1014.574,223.043,366.944,168.218,53.785,160.161
C07134=1014.567,222.795,366.969,168.214,53.794,160.162
C07135=1014.563,222.546,366.995,168.209,53.804,160.164
C07136=1014.557,222.297,367.020,168.204,53.813,160.165
C07137=1014.552,222.049,367.045,168.199,53.823,160.166
C07138=1014.547,221.800,367.069,168.196,53.833,160.167
C07139=1014.541,221.551,367.095,168.191,53.842,160.168
C07140=1014.536,221.303,367.120,168.186,53.852,160.169
C07141=1014.530,221.054,367.145,168.181,53.862,160.170
C07142=1014.525,220.805,367.170,168.177,53.871,160.171
C07143=1014.520,220.557,367.195,168.172,53.881,160.172
C07144=1014.514,220.308,367.220,168.167,53.891,160.173
C07145=1014.509,220.059,367.246,168.163,53.900,160.174
C07146=1014.504,219.812,367.270,168.159,53.910,160.176
C07147=1014.499,219.565,367.295,168.154,53.919,160.177
C07148=1014.494,219.318,367.320,168.149,53.929,160.178
C07149=1014.489,219.071,367.345,168.144,53.939,160.179
C07150=1014.484,218.824,367.370,168.140,53.948,160.180
C07151=1014.478,218.577,367.394,168.136,53.959,160.181
C07152=1014.473,218.330,367.419,168.131,53.969,160.182
C07153=1014.468,218.084,367.444,168.126,53.978,160.183
C07154=1014.463,217.835,367.469,168.123,53.988,160.185
C07155=1014.457,217.585,367.493,168.118,53.997,160.186
C07156=1014.452,217.337,367.518,168.113,54.008,160.187
C07157=1014.447,217.088,367.543,168.109,54.018,160.188
C07158=1014.442,216.840,367.567,168.104,54.027,160.189
C07159=1014.436,216.591,367.592,168.099,54.038,160.190
C07160=1014.431,216.342,367.616,168.095,54.048,160.191
C07161=1014.425,216.094,367.641,168.090,54.058,160.193
C07162=1014.420,215.845,367.666,168.085,54.068,160.194
C07163=1014.414,215.596,367.691,168.081,54.078,160.195
C07164=1014.409,215.347,367.715,168.076,54.088,160.196
C07165=1014.404,215.099,367.739,168.072,54.099,160.198
C07166=1014.399,214.850,367.764,168.067,54.108,160.199
C07167=1014.393,214.601,367.789,168.063,54.119,160.200
C07168=1014.388,214.352,367.813,168.058,54.129,160.201
C07169=1014.382,214.104,367.838,168.054,54.139,160.202
C07170=1014.377,213.855,367.862,168.049,54.149,160.203
C07171=1014.373,213.606,367.887,168.045,54.159,160.205
C07172=1014.367,213.357,367.912,168.040,54.169,160.206
C07173=1014.361,213.109,367.936,168.035,54.180,160.207
C07174=1014.356,212.860,367.960,168.031,54.190,160.208
C07175=1014.352,212.611,367.985,168.026,54.200,160.209
C07176=1014.346,212.363,368.009,168.022,54.211,160.211
C07177=1014.341,212.114,368.034,168.017,54.220,160.212
C07178=1014.336,211.865,368.058,168.013,54.231,160.213
C07179=1014.331,211.616,368.083,168.008,54.241,160.214
C07180=1014.325,211.367,368.107,168.004,54.251,160.215
C07181=1014.320,211.119,368.132,168.000,54.262,160.217
C07182=1014.315,210.870,368.156,167.995,54.272,160.218
C07183=1014.309,210.621,368.180,167.991,54.282,160.219
C07184=1014.305,210.372,368.205,167.986,54.293,160.220
C07185=1014.300,210.123,368.228,167.982,54.303,160.222
C07186=1014.294,209.875,368.253,167.977,54.313,160.223
C07187=1014.289,209.626,368.277,167.973,54.324,160.224
C07188=1014.284,209.378,368.301,167.969,54.334,160.226
C07189=1014.279,209.129,368.325,167.963,54.345,160.227
C07190=1014.274,208.880,368.350,167.959,54.355,160.228
C07191=1014.268,208.631,368.375,167.954,54.365,160.229
C07192=1014.263,208.382,368.399,167.950,54.376,160.230
C07193=1014.258,208.133,368.423,167.946,54.386,160.232
C07194=1014.253,207.884,368.447,167.942,54.397,160.233
C07195=1014.248,207.635,368.471,167.936,54.408,160.234
C07196=1014.242,207.387,368.495,167.932,54.418,160.236
C07197=1014.237,207.138,368.519,167.928,54.429,160.237
C07198=1014.232,206.889,368.543,167.924,54.440,160.238
C07199=1014.227,206.640,368.567,167.919,54.450,160.239
C07200=1014.221,206.392,368.591,167.914,54.461,160.241
C07201=1014.215,206.143,368.615,167.910,54.472,160.242
C07202=1014.210,205.894,368.638,167.906,54.482,160.243
C07203=1014.205,205.646,368.663,167.901,54.493,160.245
C07204=1014.200,205.396,368.686,167.896,54.504,160.246
C07205=1014.195,205.148,368.710,167.892,54.514,160.247
C07206=1014.190,204.913,368.733,167.887,54.524,160.248
C07207=1014.185,204.677,368.755,167.884,54.534,160.250
C07208=1014.180,204.443,368.778,167.880,54.545,160.251
C07209=1014.175,204.207,368.800,167.875,54.555,160.252
C07210=1014.171,203.972,368.822,167.871,54.565,160.253
C07211=1014.166,203.737,368.845,167.866,54.575,160.254
C07212=1014.161,203.502,368.867,167.863,54.585,160.256
C07213=1014.156,203.267,368.890,167.859,54.596,160.257
C07214=1014.137,202.159,368.988,167.332,54.506,160.118
C07215=1014.133,201.910,369.010,167.327,54.518,160.120
C07216=1014.128,201.662,369.032,167.321,54.530,160.121
C07217=1014.124,201.412,369.054,167.316,54.542,160.122
C07218=1014.120,201.163,369.076,167.312,54.554,160.124
C07219=1014.116,200.914,369.098,167.307,54.566,160.125
C07220=1014.112,200.665,369.120,167.303,54.577,160.127
C07221=1014.108,200.416,369.143,167.298,54.589,160.128
C07222=1014.104,200.167,369.164,167.293,54.600,160.129
C07223=1014.099,199.918,369.186,167.289,54.612,160.131
C07224=1014.096,199.669,369.208,167.284,54.625,160.132
C07225=1014.091,199.421,369.230,167.279,54.636,160.133
C07226=1014.087,199.171,369.252,167.275,54.648,160.135
C07227=1014.084,198.922,369.274,167.270,54.660,160.136
C07228=1014.079,198.673,369.295,167.265,54.672,160.137
C07229=1014.075,198.424,369.317,167.261,54.684,160.139
C07230=1014.071,198.174,369.339,167.256,54.696,160.140
C07231=1014.067,197.926,369.360,167.251,54.708,160.142
C07232=1014.062,197.677,369.381,167.247,54.720,160.143
C07233=1014.058,197.428,369.404,167.242,54.732,160.145
C07234=1014.054,197.179,369.425,167.237,54.744,160.146
C07235=1014.049,196.930,369.447,167.233,54.756,160.148
C07236=1014.045,196.681,369.468,167.228,54.768,160.149
C07237=1014.042,196.432,369.489,167.223,54.780,160.150
C07238=1014.037,196.183,369.511,167.219,54.792,160.152
C07239=1014.032,195.933,369.532,167.214,54.804,160.153
C07240=1014.028,195.685,369.554,167.209,54.816,160.154
C07241=1014.024,195.436,369.575,167.205,54.828,160.156
C07242=1014.020,195.186,369.596,167.200,54.840,160.157
C07243=1014.015,194.938,369.618,167.196,54.852,160.159
C07244=1014.012,194.688,369.640,167.191,54.863,160.160
C07245=1014.007,194.439,369.661,167.187,54.876,160.162
C07246=1014.003,194.191,369.682,167.182,54.888,160.163
C07247=1013.998,193.941,369.704,167.177,54.900,160.164
C07248=1013.995,193.692,369.725,167.173,54.912,160.166
C07249=1013.990,193.443,369.747,167.168,54.924,160.167
C07250=1013.986,193.194,369.768,167.163,54.936,160.169
C07251=1013.982,192.945,369.789,167.159,54.947,160.170
C07252=1013.978,192.695,369.810,167.155,54.960,160.172
C07253=1013.974,192.447,369.832,167.151,54.971,160.173
C07254=1013.969,192.198,369.853,167.146,54.983,160.174
C07255=1013.966,191.949,369.874,167.141,54.995,160.176
C07256=1013.962,191.699,369.896,167.137,55.008,160.177
C07257=1013.958,191.451,369.916,167.132,55.019,160.179
C07258=1013.953,191.202,369.938,167.127,55.031,160.180
C07259=1013.950,190.953,369.960,167.124,55.043,160.181
C07260=1013.945,190.703,369.981,167.120,55.055,160.183
C07261=1013.941,190.455,370.002,167.115,55.067,160.184
C07262=1013.937,190.205,370.023,167.110,55.079,160.186
C07263=1013.933,189.957,370.045,167.105,55.091,160.187
C07264=1013.929,189.707,370.066,167.101,55.103,160.189
C07265=1013.925,189.459,370.087,167.098,55.115,160.190
C07266=1013.921,189.209,370.108,167.093,55.127,160.192
C07267=1013.917,188.960,370.129,167.088,55.138,160.193
C07268=1013.913,188.711,370.150,167.084,55.151,160.195
C07269=1013.909,188.462,370.171,167.080,55.162,160.196
